	30: (* wait for com cycle *)
		IF NOT StartJob(TRUE) THEN // Not Busy, Execute set to True
			IF Error
			THEN
				ErrorText									:= CONCAT('Error at SlaveNo: ',	CONCAT(INT_TO_STRING(SlaveNo), CONCAT(', JobNo: ', INT_TO_STRING(JobNo))));
				SlaveCom[SlaveNo]^.countBad 				:= SlaveCom[SlaveNo]^.countBad +1;
				SlaveInErrorMask							:= CSETBIT32(SlaveInErrorMask,TO_SINT(SlaveNo),TRUE);
				IF Options.0
				THEN
					JobNo 									:= JobNo + 1;
					state 									:= 10;	(* next job *)				
				ELSE
					state 									:= 98; 					
				END_IF
			ELSE
				SlaveInErrorMask							:= CSETBIT32(SlaveInErrorMask,TO_SINT(SlaveNo),FALSE);
				SlaveCom[SlaveNo]^.countGood 				:= SlaveCom[SlaveNo]^.countGood +1;
				SlaveCom[SlaveNo]^.Jobs[JobNo].Valid 		:= TRUE;
				SlaveCom[SlaveNo]^.Jobs[JobNo].TimeStamp 	:= Timestamp;
				JobNo 										:= JobNo + 1;
				state 										:= 10;	(* next job *)
			END_IF
			StartJob(FALSE);
		END_IF

	98: (* wait for quit *)
		;


	END_CASE

METHOD PRIVATE getNextJob : Bool //Return value = TRUE if execution finished
VAR_INPUT
END_VAR
	
	WHILE SlaveCom[SlaveNo]^.Jobs[JobNo].FunctionCode = 0 DO
		JobNo 											:= JobNo + 1;
		IF JobNo > SlaveCom[SlaveNo]^.MAX_SLAVE_JOB THEN
			JobNo 										:= SlaveCom[SlaveNo]^.MIN_SLAVE_JOB;
			SlaveNo 									:= SlaveNo + 1;
			GetNextJob									:= FALSE;
			RETURN;
		END_IF
	END_WHILE
	GetNextJob											:= TRUE;
END_METHOD

METHOD PRIVATE getNextSlave : Bool //Return value = TRUE if execution finished
VAR_INPUT
END_VAR
	WHILE SlaveCom[SlaveNo] = 0 OR_ELSE NOT SlaveCom[SlaveNo]^.Enable DO
		SlaveNo 										:= SlaveNo + 1;
		IF SlaveNo > MAX_SLAVE 
		THEN
			k 											:= k + 1;
			SlaveNo 									:= MIN_SLAVE;
		ELSIF k = 2 
		THEN
			k 											:= 0;
			GetNextSlave								:= FALSE;
			RETURN;
		END_IF	
	END_WHILE
	GetNextSlave										:= TRUE;
END_METHOD

METHOD PUBLIC reset : BOOL //Return value = TRUE if execution finished
VAR_INPUT
END_VAR
IF State = 98 
THEN
	state													:= 0;
END_IF
Error														:= FALSE;
ErrorID														:= 0;
ErrorText													:= '';
reset														:= TRUE;
END_METHOD

METHOD PRIVATE startJob : BOOL //Return value = TRUE if busy - TRUE as long as the job is busy
VAR_INPUT
	Execute							: BOOL;
END_VAR
(* ModbusCOM Baustein mit parametern antriggern *)
	IF 	SlaveCom[SlaveNo]^.Jobs[JobNo].FunctionCode = 1 THEN
		com.ReadCoils(
			UnitID			:= SlaveCom[SlaveNo]^.Address,					(*UnitID: Modbus Stationsadresse (1..247). Der Modbus-Slave antwortet nur, wenn er Telegramme mit seiner eigenen Stationsadresse empfängt. optional können hier auch Sammeladressen eingestellt werden um auf beliebige Anfragen zu antworten. Die Adresse 0 ist für Broadcast-Telegramme reserviert und somit keine gültige Stationsadresse.*)
			Quantity		:= SlaveCom[SlaveNo]^.jobs[JobNo].Quantity,		(*Quantity: Anzahl der zu lesenden oder zu schreibenden Datenworte bei Wort-orientierten Modbus-Funktionen. Bei Bit-orientierten Modbus-Funktionen gibt Quantity die Anzahl der Bits (Inputs oder Coils) an.*)
			MBAddr			:= SlaveCom[SlaveNo]^.jobs[JobNo].startAddress,	(*MBAddr: Modbus-Datenadresse, von der die Daten aus dem Endgerät (Slave) gelesen werden. Diese Adresse wird unverändert zum Slave übertragen und wird dort als Datenadresse interpretiert.*)
			cbLength		:= SlaveCom[SlaveNo]^.jobs[JobNo].Quantity, 	(*cbLength : Größe der verwendeten Datenvariable für Sende- oder Lese-Aktionen in Bytes. cbLength muss größer oder gleich der durch Quantity bestimmten übertragenen Datenmenge sein. Bei Wortzugriffen gilt z. B.: [cbLength >= Quantity * 2]. cbLength kann mit SIZEOF(ModbusDaten) berechnet werden.*)
			pMemoryAddr		:= ADR(SlaveCom[SlaveNo]^.Data),				(*pMemoryAddr: Speicheradresse in der SPS, die mit ADR(ModbusDaten) berechnet wird. Bei Leseaktionen werden die gelesenen Daten in der adressierten Variablen abgelegt. Bei Sende-Aktionen werden die Daten aus der adressierten Variablen zum Endgerät übertragen.*)
			Execute			:= Execute,
			Timeout			:= ,
			BUSY			=> StartJob,									(*Busy: Zeigt an, dass der Funktionsbaustein aktiv ist. Busy wird mit steigender Flanke an Execute TRUE und wird wieder FALSE nachdem die gestartete Aktion beendet ist. Es kann immer nur eine Aktion gleichzeitig aktiv sein.*)
			Error			=> Error,										(*Error: Zeigt an, dass bei der Bearbeitung einer Aktion ein Fehler aufgetreten ist*)
			ErrorId			=> ErrorID);									(*ErrorId: Zeigt eine Fehlernummer im Falle einer gestörten oder fehlerhaften Kommunikation an.*)	

	ELSIF 	SlaveCom[SlaveNo]^.Jobs[JobNo].FunctionCode = 3 THEN
		com.ReadRegs(
			UnitID			:= SlaveCom[SlaveNo]^.Address,		
			Quantity		:= SlaveCom[SlaveNo]^.jobs[JobNo].Quantity,
			MBAddr			:= SlaveCom[SlaveNo]^.jobs[JobNo].startAddress,
			cbLength		:= SlaveCom[SlaveNo]^.jobs[JobNo].Quantity * 2,
			pMemoryAddr		:= ADR(SlaveCom[SlaveNo]^.data),
			Execute			:= Execute,
			Timeout			:= ,
			BUSY			=> StartJob,
			Error			=> Error,
			ErrorId			=> ErrorID);
	
	ELSIF 	SlaveCom[SlaveNo]^.Jobs[JobNo].FunctionCode = 4 THEN
		com.ReadInputRegs(
			UnitID			:= SlaveCom[SlaveNo]^.Address,		
			Quantity		:= SlaveCom[SlaveNo]^.jobs[JobNo].Quantity,
			MBAddr			:= SlaveCom[SlaveNo]^.jobs[JobNo].startAddress,
			cbLength		:= SlaveCom[SlaveNo]^.jobs[JobNo].Quantity * 2,
			pMemoryAddr		:= ADR(SlaveCom[SlaveNo]^.data),
			Execute			:= Execute,
			Timeout			:= ,
			BUSY			=> StartJob,
			Error			=> Error,
			ErrorId			=> ErrorID);
	
	ELSIF 	SlaveCom[SlaveNo]^.Jobs[JobNo].FunctionCode = 5 THEN
		com.WriteSingleCoil(
			UnitID			:= SlaveCom[SlaveNo]^.Address,		
			Quantity		:= SlaveCom[SlaveNo]^.jobs[JobNo].Quantity,
			MBAddr			:= SlaveCom[SlaveNo]^.jobs[JobNo].startAddress,
			cbLength		:= SlaveCom[SlaveNo]^.jobs[JobNo].Quantity,
			pMemoryAddr		:= ADR(SlaveCom[SlaveNo]^.data),
			Execute			:= Execute,
			Timeout			:= ,
			BUSY			=> StartJob,
			Error			=> Error,
			ErrorId			=> ErrorID);
			
	ELSIF 	SlaveCom[SlaveNo]^.Jobs[JobNo].FunctionCode = 6 THEN
		com.WriteSingleRegister(
			UnitID			:= SlaveCom[SlaveNo]^.Address,		
			Quantity		:= SlaveCom[SlaveNo]^.jobs[JobNo].Quantity,
			MBAddr			:= SlaveCom[SlaveNo]^.jobs[JobNo].startAddress,
			cbLength		:= SlaveCom[SlaveNo]^.jobs[JobNo].Quantity,
			pMemoryAddr		:= ADR(SlaveCom[SlaveNo]^.data),
			Execute			:= Execute,
			Timeout			:= ,
			BUSY			=> StartJob,
			Error			=> Error,
			ErrorId			=> ErrorID);
		
	ELSIF 	SlaveCom[SlaveNo]^.Jobs[JobNo].FunctionCode = 8 THEN
		com.Diagnostics(
			UnitID			:= SlaveCom[SlaveNo]^.Address,		
			Quantity		:= SlaveCom[SlaveNo]^.jobs[JobNo].Quantity,
			MBAddr			:= SlaveCom[SlaveNo]^.jobs[JobNo].startAddress,
			cbLength		:= SlaveCom[SlaveNo]^.jobs[JobNo].Quantity,
			pMemoryAddr		:= ADR(SlaveCom[SlaveNo]^.data),
			Execute			:= Execute,
			Timeout			:= ,
			BUSY			=> StartJob,
			Error			=> Error,
			ErrorId			=> ErrorID);
		
	ELSIF 	SlaveCom[SlaveNo]^.Jobs[JobNo].FunctionCode = 15 THEN
		com.WriteMultipleCoils(
			UnitID			:= SlaveCom[SlaveNo]^.Address,		
			Quantity		:= SlaveCom[SlaveNo]^.jobs[JobNo].Quantity,
			MBAddr			:= SlaveCom[SlaveNo]^.jobs[JobNo].startAddress,
			cbLength		:= SlaveCom[SlaveNo]^.jobs[JobNo].Quantity,
			pMemoryAddr		:= ADR(SlaveCom[SlaveNo]^.data),
			Execute			:= Execute,
			Timeout			:= ,
			BUSY			=> StartJob,
			Error			=> Error,
			ErrorId			=> ErrorID);
	
	ELSIF 	SlaveCom[SlaveNo]^.Jobs[JobNo].FunctionCode = 16 THEN
		com.WriteRegs(
			UnitID			:= SlaveCom[SlaveNo]^.Address,		
			Quantity		:= SlaveCom[SlaveNo]^.jobs[JobNo].Quantity,
			MBAddr			:= SlaveCom[SlaveNo]^.jobs[JobNo].startAddress,
			cbLength		:= SlaveCom[SlaveNo]^.jobs[JobNo].Quantity,
			pMemoryAddr		:= ADR(SlaveCom[SlaveNo]^.data),
			Execute			:= Execute,
			Timeout			:= ,
			BUSY			=> StartJob,
			Error			=> Error,
			ErrorId			=> ErrorID);
			
	END_IF
END_METHOD

END_FUNCTION_BLOCK

// ---- POUs/Connectivity/TF625x-Modbus/Master/TF6255-ModbusRtu/ModbusRtuMaster5B.TcPOU
{attribute 'no_check'}
// ModBus comunication master to multible slaves useing RTU protocol
// based on TF6255 - required lib: Tc2_ModbusRTU
FUNCTION_BLOCK ModbusRtuMaster5B
VAR_OUTPUT CONSTANT
	MIN_SLAVE												:	INT := 1;
	MAX_SLAVE												:	INT := PARAM.MODBUS_MAX_SLAVES_OF_MASTER;
{attribute 'displaymode':='binary'}
	OPTION_DISABLE_ERROR_STATE								:	BYTE := 2#0000_0001; //FB will not go into error state and keeps running, even all slaves are in error state
END_VAR
VAR_INPUT
	Enable													:	BOOL ; 		// FB will be processed as long as enable is TRUE 
	ResetTrig												:	BOOL ;		// The function block will be reset with a rising edge 
{attribute 'displaymode':='binary'}
	Options													:	BYTE := 0; //FB options, see VAR_OUTPUT CONSTANT
	SlaveCom												:	ARRAY[MIN_SLAVE..MAX_SLAVE] OF POINTER TO ModbusSlaveCom;
	Timestamp												:	DT;
END_VAR         	
VAR_OUTPUT     
	JobNo													:	INT := 0;
	SlaveNo													:	INT := 0;
{attribute 'displaymode':='binary'}
	SlaveInErrorMask										:	DWORD; //Bit.1 indicates slave 1 in error 	
	Error													:	BOOL;		// Rising edge of Error informs that an error occurred during the execution of the Function Block 
{attribute 'displaymode':='hex'}
	ErrorID													:	MODBUS_ERRORS;		// Error identification - see ADS return codes at Beckhoff infosys for further information 
	ErrorText												:	STRING;
END_VAR
VAR
(* memory **************************************************)
	State 													:	INT := 0;

(* trigger *************************************************)

(* timer ***************************************************)

(* blocks **************************************************)
//	com														:	ModbusRtuMaster_PcCOM := (Timeout := DEFAULT_ADS_TIMEOUT);
//	com														:	ModbusRtuMaster_KL6x22B := (Timeout := DEFAULT_ADS_TIMEOUT);
	com														:	ModbusRtuMaster_KL6x5B := (Timeout := DEFAULT_ADS_TIMEOUT);
(* internal used variables *********************************)
	i,j,k													:	INT :=0;
END_VAR

(* ModBus RTU comunication to multible slaves 	JHue V1.0			*)
(* uncomment necessary master funktion block 						*)
(* use TC2_ModBusRTU.lib											*)
(********************************************************************)
	IF ResetTrig THEN
		reset();
	END_IF
	
	CASE state OF
	0:	(* Idle *)
		IF Enable 
		THEN
			k 												:=	0;
			JobNo  :=  SlaveNo								:=	1;
			state 											:=	10;
		END_IF

	10: 
		IF GetNextSlave() 
		THEN (* find Slave *)
			k 												:= 0;
			IF GetNextJob() 
			THEN (* find JobNo *)
				SlaveCom[SlaveNo]^.currentJobIdx 			:= JobNo;
				SlaveCom[SlaveNo]^.writeJobRequested 		:= SlaveCom[SlaveNo]^.Jobs[JobNo].FunctionCode >= 5;
				State 										:= SEL(SlaveCom[SlaveNo]^.writeJobRequested, 20, 15);
			END_IF
		ELSE
			state 											:=	0;
		END_IF
	
	15: (* wait for valid write date *)
		IF NOT SlaveCom[SlaveNo]^.writeJobRequested
		THEN
			SlaveCom[SlaveNo]^.Jobs[JobNo].Valid 			:= FALSE;
			state 											:= 20;
		END_IF

	20: (* start job *)	
		IF NOT StartJob(FALSE) // Busy
		THEN						
			state 											:= 30;
		END_IF

	30: (* wait for com cycle *)
		IF NOT StartJob(TRUE) THEN // Not Busy, Execute set to True
			IF Error
			THEN
				ErrorText									:= CONCAT('Error at SlaveNo: ',	CONCAT(INT_TO_STRING(SlaveNo), CONCAT(', JobNo: ', INT_TO_STRING(JobNo))));
				SlaveCom[SlaveNo]^.countBad 				:= SlaveCom[SlaveNo]^.countBad +1;
				SlaveInErrorMask							:= CSETBIT32(SlaveInErrorMask,TO_SINT(SlaveNo),TRUE);
				IF Options.0
				THEN
					JobNo 									:= JobNo + 1;
					state 									:= 10;	(* next job *)				
				ELSE
					state 									:= 98; 					
				END_IF
			ELSE
				SlaveInErrorMask							:= CSETBIT32(SlaveInErrorMask,TO_SINT(SlaveNo),FALSE);
				SlaveCom[SlaveNo]^.countGood 				:= SlaveCom[SlaveNo]^.countGood +1;
				SlaveCom[SlaveNo]^.Jobs[JobNo].Valid 		:= TRUE;
				SlaveCom[SlaveNo]^.Jobs[JobNo].TimeStamp 	:= Timestamp;
				JobNo 										:= JobNo + 1;
				state 										:= 10;	(* next job *)
			END_IF
			StartJob(FALSE);
		END_IF

	98: (* wait for quit *)
		;


	END_CASE

METHOD PRIVATE getNextJob : Bool
VAR_INPUT
END_VAR
	
	WHILE SlaveCom[SlaveNo]^.Jobs[JobNo].FunctionCode = 0 DO
		JobNo 											:= JobNo + 1;
		IF JobNo > SlaveCom[SlaveNo]^.MAX_SLAVE_JOB THEN
			JobNo 										:= SlaveCom[SlaveNo]^.MIN_SLAVE_JOB;
			SlaveNo 									:= SlaveNo + 1;
			GetNextJob									:= FALSE;
			RETURN;
		END_IF
	END_WHILE
	GetNextJob											:= TRUE;
END_METHOD

METHOD PRIVATE getNextSlave : Bool
VAR_INPUT
END_VAR
	WHILE SlaveCom[SlaveNo] = 0 OR_ELSE NOT SlaveCom[SlaveNo]^.Enable DO
		SlaveNo 										:= SlaveNo + 1;
		IF SlaveNo > MAX_SLAVE 
		THEN
			k 											:= k + 1;
			SlaveNo 									:= MIN_SLAVE;
		ELSIF k = 2 
		THEN
			k 											:= 0;
			GetNextSlave								:= FALSE;
			RETURN;
		END_IF	
	END_WHILE
	GetNextSlave										:= TRUE;
END_METHOD

METHOD PUBLIC reset : booL //Return value = TRUE if execution finished
VAR_INPUT
END_VAR
IF State = 98 
THEN
	state													:= 0;
END_IF
Error														:= FALSE;
ErrorID														:= 0;
ErrorText													:= '';
reset														:= TRUE;
END_METHOD

METHOD PRIVATE startJob : BOOL //Return value = TRUE if busy - TRUE as long as the job is busy
VAR_INPUT
	Execute							: BOOL;
END_VAR
(* ModbusCOM Baustein mit parametern antriggern *)
	IF 		SlaveCom[SlaveNo]^.Jobs[JobNo].FunctionCode = 1 THEN
		com.ReadCoils(
			UnitID			:= SlaveCom[SlaveNo]^.Address,				(*UnitID: Modbus Stationsadresse (1..247). Der Modbus-Slave antwortet nur, wenn er Telegramme mit seiner eigenen Stationsadresse empfängt. optional können hier auch Sammeladressen eingestellt werden um auf beliebige Anfragen zu antworten. Die Adresse 0 ist für Broadcast-Telegramme reserviert und somit keine gültige Stationsadresse.*)
			Quantity		:= SlaveCom[SlaveNo]^.jobs[JobNo].Quantity,		(*Quantity: Anzahl der zu lesenden oder zu schreibenden Datenworte bei Wort-orientierten Modbus-Funktionen. Bei Bit-orientierten Modbus-Funktionen gibt Quantity die Anzahl der Bits (Inputs oder Coils) an.*)
			MBAddr			:= SlaveCom[SlaveNo]^.jobs[JobNo].startAddress,	(*MBAddr: Modbus-Datenadresse, von der die Daten aus dem Endgerät (Slave) gelesen werden. Diese Adresse wird unverändert zum Slave übertragen und wird dort als Datenadresse interpretiert.*)
			cbLength		:= SlaveCom[SlaveNo]^.jobs[JobNo].Quantity, 	(*cbLength : Größe der verwendeten Datenvariable für Sende- oder Lese-Aktionen in Bytes. cbLength muss größer oder gleich der durch Quantity bestimmten übertragenen Datenmenge sein. Bei Wortzugriffen gilt z. B.: [cbLength >= Quantity * 2]. cbLength kann mit SIZEOF(ModbusDaten) berechnet werden.*)
			pMemoryAddr		:= ADR(SlaveCom[SlaveNo]^.Data),				(*pMemoryAddr: Speicheradresse in der SPS, die mit ADR(ModbusDaten) berechnet wird. Bei Leseaktionen werden die gelesenen Daten in der adressierten Variablen abgelegt. Bei Sende-Aktionen werden die Daten aus der adressierten Variablen zum Endgerät übertragen.*)
			Execute			:= Execute,
			Timeout			:= ,
			BUSY			=> StartJob,									(*Busy: Zeigt an, dass der Funktionsbaustein aktiv ist. Busy wird mit steigender Flanke an Execute TRUE und wird wieder FALSE nachdem die gestartete Aktion beendet ist. Es kann immer nur eine Aktion gleichzeitig aktiv sein.*)
			Error			=> Error,										(*Error: Zeigt an, dass bei der Bearbeitung einer Aktion ein Fehler aufgetreten ist*)
			ErrorId			=> ErrorID);									(*ErrorId: Zeigt eine Fehlernummer im Falle einer gestörten oder fehlerhaften Kommunikation an.*)	
	
	ELSIF 	SlaveCom[SlaveNo]^.Jobs[JobNo].FunctionCode = 3 THEN
		com.ReadRegs(
			UnitID			:= SlaveCom[SlaveNo]^.Address,		
			Quantity		:= SlaveCom[SlaveNo]^.jobs[JobNo].Quantity,
			MBAddr			:= SlaveCom[SlaveNo]^.jobs[JobNo].startAddress,
			cbLength		:= SlaveCom[SlaveNo]^.jobs[JobNo].Quantity * 2,
			pMemoryAddr		:= ADR(SlaveCom[SlaveNo]^.data),
			Execute			:= Execute,
			Timeout			:= ,
			BUSY			=> StartJob,
			Error			=> Error,
			ErrorId			=> ErrorID);
	
	ELSIF 	SlaveCom[SlaveNo]^.Jobs[JobNo].FunctionCode = 4 THEN
		com.ReadInputRegs(
			UnitID			:= SlaveCom[SlaveNo]^.Address,		
			Quantity		:= SlaveCom[SlaveNo]^.jobs[JobNo].Quantity,
			MBAddr			:= SlaveCom[SlaveNo]^.jobs[JobNo].startAddress,
			cbLength		:= SlaveCom[SlaveNo]^.jobs[JobNo].Quantity * 2,
			pMemoryAddr		:= ADR(SlaveCom[SlaveNo]^.data),
			Execute			:= Execute,
			Timeout			:= ,
			BUSY			=> StartJob,
			Error			=> Error,
			ErrorId			=> ErrorID);
	
	ELSIF 	SlaveCom[SlaveNo]^.Jobs[JobNo].FunctionCode = 5 THEN
		com.WriteSingleCoil(
			UnitID			:= SlaveCom[SlaveNo]^.Address,		
			Quantity		:= SlaveCom[SlaveNo]^.jobs[JobNo].Quantity,
			MBAddr			:= SlaveCom[SlaveNo]^.jobs[JobNo].startAddress,
			cbLength		:= SlaveCom[SlaveNo]^.jobs[JobNo].Quantity,
			pMemoryAddr		:= ADR(SlaveCom[SlaveNo]^.data),
			Execute			:= Execute,
			Timeout			:= ,
			BUSY			=> StartJob,
			Error			=> Error,
			ErrorId			=> ErrorID);
		
	ELSIF 	SlaveCom[SlaveNo]^.Jobs[JobNo].FunctionCode = 6 THEN
		com.WriteSingleRegister(
			UnitID			:= SlaveCom[SlaveNo]^.Address,		
			Quantity		:= SlaveCom[SlaveNo]^.jobs[JobNo].Quantity,
			MBAddr			:= SlaveCom[SlaveNo]^.jobs[JobNo].startAddress,
			cbLength		:= SlaveCom[SlaveNo]^.jobs[JobNo].Quantity,
			pMemoryAddr		:= ADR(SlaveCom[SlaveNo]^.data),
			Execute			:= Execute,
			Timeout			:= ,
			BUSY			=> StartJob,
			Error			=> Error,
			ErrorId			=> ErrorID);
			
	ELSIF 	SlaveCom[SlaveNo]^.Jobs[JobNo].FunctionCode = 8 THEN
		com.Diagnostics(
			UnitID			:= SlaveCom[SlaveNo]^.Address,		
			Quantity		:= SlaveCom[SlaveNo]^.jobs[JobNo].Quantity,
			MBAddr			:= SlaveCom[SlaveNo]^.jobs[JobNo].startAddress,
			cbLength		:= SlaveCom[SlaveNo]^.jobs[JobNo].Quantity,
			pMemoryAddr		:= ADR(SlaveCom[SlaveNo]^.data),
			Execute			:= Execute,
			Timeout			:= ,
			BUSY			=> StartJob,
			Error			=> Error,
			ErrorId			=> ErrorID);
	
	ELSIF 	SlaveCom[SlaveNo]^.Jobs[JobNo].FunctionCode = 15 THEN
		com.WriteMultipleCoils(
			UnitID			:= SlaveCom[SlaveNo]^.Address,		
			Quantity		:= SlaveCom[SlaveNo]^.jobs[JobNo].Quantity,
			MBAddr			:= SlaveCom[SlaveNo]^.jobs[JobNo].startAddress,
			cbLength		:= SlaveCom[SlaveNo]^.jobs[JobNo].Quantity,
			pMemoryAddr		:= ADR(SlaveCom[SlaveNo]^.data),
			Execute			:= Execute,
			Timeout			:= ,
			BUSY			=> StartJob,
			Error			=> Error,
			ErrorId			=> ErrorID);
	
	ELSIF 	SlaveCom[SlaveNo]^.Jobs[JobNo].FunctionCode = 16 THEN
		com.WriteRegs(
			UnitID			:= SlaveCom[SlaveNo]^.Address,		
			Quantity		:= SlaveCom[SlaveNo]^.jobs[JobNo].Quantity,
			MBAddr			:= SlaveCom[SlaveNo]^.jobs[JobNo].startAddress,
			cbLength		:= SlaveCom[SlaveNo]^.jobs[JobNo].Quantity,
			pMemoryAddr		:= ADR(SlaveCom[SlaveNo]^.data),
			Execute			:= Execute,
			Timeout			:= ,
			BUSY			=> StartJob,
			Error			=> Error,
			ErrorId			=> ErrorID);	
	END_IF
END_METHOD

END_FUNCTION_BLOCK

// ---- POUs/Connectivity/TF6310-TcpServer/TcpBasic/TCPSendRecCtrl.TcPOU
{attribute 'no_check'}
//Send or receive data via TCP connection 
//based on TF6310, required lib: Tc2_TcpIp - see Beckhoff Infosys for more information
FUNCTION_BLOCK TCPSendRecCtrl EXTENDS FbBase
VAR_OUTPUT CONSTANT
	FNC_RECEIVE												:	INT := 0;
	FNC_SEND												:	INT := 1;
END_VAR                 									
VAR_INPUT               									
	Fnc														:	INT (FNC_RECEIVE..FNC_SEND) := FNC_RECEIVE;
	SrvNetId												: 	T_AmsNetId := ''; (* server ams net id *)
	Timeout													: 	TIME := DEFAULT_ADS_TIMEOUT; //ADS timeout
{attribute 'displaymode':='binary'}
	Options													:	BYTE := 2#0000_0000; //Options Bit .0 = Do NOT restart receive internally
	hSocket													:	T_HSOCKET; //Server handle
	pData													:	POINTER TO BYTE; //Pointer do send/res data field 
	cbData													:	UDINT; //Size of send/rec data field 
	EnableDebugMode											:	BOOL; //Write debug information into twincat logger
END_VAR
VAR_OUTPUT
	RecBytes 												:  UDINT;  	// Count of received bytes
	WinsockErrorId											:	E_WinsockError;  //Winsocket error enum - see TF6310 documentation for further information
END_VAR
VAR
(* cache ************************************************************)
	MemFnc													:	INT := -1;

(* function-block instances ***************************************************************)
	SocketSend												:	FB_SocketSend;
	SocketReceive											:	FB_SocketReceive;

END_VAR


(* Execute ***************************************************************************************)
	rtExecute(CLK := Execute);
	IF rtExecute.Q
		AND MemFnc < 0
	THEN
		MemFnc 												:= SEL(Fnc = FNC_SEND, FNC_RECEIVE , FNC_SEND) ;
		Busy												:= TRUE;
		Done												:= FALSE;
		Error												:= FALSE;
		ErrorID												:= 0;
	END_IF

(* Call Method ***********************************************************************************)
	CASE MemFnc OF
	FNC_SEND:
		SEND(Execute:= Execute);

	FNC_RECEIVE:
		Receive(Execute	:= Execute);

	-1:
		IF NOT Execute
		THEN
			Busy											:= FALSE;
			Done											:= FALSE;
			Error											:= FALSE;
			ErrorID											:= 0;
		END_IF                              				
	ELSE                                    				
		Busy												:= FALSE;
		Done												:= FALSE;
		Error												:= Execute;
		ErrorID												:= E_AdsErr.DEVICE_INVALIDPARM;
	END_CASE

(*************************************************************************************************)

PROPERTY PUBLIC optDoNotRestartReceiveCyclic : BOOL
GET
optDoNotRestartReceiveCyclic := Options.0;
END_GET
SET
Options.0 := optDoNotRestartReceiveCyclic;
END_SET
END_PROPERTY

METHOD PUBLIC receive : BOOL //Return value = TRUE if busy
//required parameter
//hSocket
//pData
//cbData
VAR_INPUT
	Execute													:	BOOL;
END_VAR
	MemFnc													:= FNC_RECEIVE;
	THIS^.Execute											:= Execute;
	                                						
IF pData = 0                        						
THEN                                						
	Busy													:= NOT Error;
	Error													:= TRUE;
	ErrorId													:= E_AdsErr.DEVICE_INVALIDPARM;
	Done													:= FALSE;
	MemFnc													:= SEL(Execute , -1 ,MemFnc); 
	RETURN;                         	
END_IF

	IF Execute
	THEN
		Error												:=	FALSE;
		ErrorId												:= 0;
		SocketReceive.bExecute 								:= TRUE;
	ELSIF NOT SocketReceive.bBusy   						
	THEN                            						
		Error												:=	FALSE;
		ErrorId												:= 0;
		SocketReceive.bExecute 								:= FALSE;
	END_IF                          	
                                    	
	SocketReceive(
			sSrvNetId	:= SrvNetId,
			hSocket		:= hSocket,
			cbLen		:= cbData,
			pDest		:= pData,
			bExecute	:= ,
			tTimeout	:= Timeout,
			bBusy		=> Busy,
			bError		=> ,
			nErrId		=> ,
			nRecBytes	=> );

	IF NOT SocketReceive.bBusy
		AND NOT SocketReceive.bError
		AND SocketReceive.bExecute
	THEN
		IF EnableDebugMode
			AND SocketReceive.nRecBytes > 0
			AND NOT Done
		THEN
			ADSLOGDINT(	ADSLOG_MSGTYPE_ERROR OR ADSLOG_MSGTYPE_LOG, CONCAT('%d Bytes received / ', HSOCKET_TO_STRING(hSocket)) , UDINT_TO_DINT(SocketReceive.nRecBytes));
		END_IF
		Done												:= SocketReceive.nRecBytes > 0 OR Options.0; (* Done melden nach jedenm Lesezyklus, egal ob Daten empfangen wurden *)
		IF NOT Done
		THEN (* only set Done if something is safely received *)
			SocketReceive(bExecute := FALSE);
			SocketReceive(bExecute := TRUE, bBusy => Busy);
		END_IF
		RecBytes											:= SEL(Done , 0 ,SocketReceive.nRecBytes);
	ELSE                                					
		Done												:= FALSE;
	END_IF                              	
                                        	
	IF NOT Busy
	THEN
		IF SocketReceive.bExecute
		THEN
			Error											:=	SocketReceive.bError;
			IF SocketReceive.nErrId >= 16#80070000
			THEN
				ErrorId										:= E_ADSERR.CLIENT_W32ERROR;
				WinsockErrorId								:= ADSERROR_TO_WSERROR(SocketReceive.nErrId);
			ELSE                    						
				ErrorId										:= SocketReceive.nErrId;
				WinsockErrorId								:= WSOK;
			END_IF
		END_IF
		IF NOT Execute
		THEN
			MemFnc											:= -1;
			SocketReceive(bExecute := FALSE);
		END_IF
	END_IF
	
	//Method return
	Receive													:= Busy;
END_METHOD

METHOD PUBLIC send : BOOL //Return value = TRUE if busy
//required parameter
//hSocket
//pData
//cbData
VAR_INPUT
	Execute													:	BOOL;
END_VAR
	MemFnc													:= FNC_SEND;
	THIS^.Execute											:= Execute;
	
IF pData = 0 THEN
	Busy													:= NOT Error;
	Error													:= TRUE;
	ErrorId													:= E_ADSErr.DEVICE_INVALIDPARM;
	Done													:= FALSE;
	MemFnc													:= SEL(Execute , -1 ,MemFnc); 
	RETURN;
END_IF

	IF Execute
	THEN
		Error												:=	FALSE;
		ErrorId												:= 0;
		SocketSend.bExecute 								:= TRUE;
	ELSIF NOT SocketSend.bBusy          					
	THEN                                					
		Error												:=	FALSE;
		ErrorId												:= 0;
		SocketSend.bExecute 								:= FALSE;
	END_IF                              	
	                                    	
	SocketSend(
		sSrvNetId	:= SrvNetId,
		hSocket		:= hSocket,
		cbLen		:= cbData,
		pSrc		:= pData,
		bExecute	:= ,
		tTimeout	:= Timeout,
		bBusy		=> Busy,
		bError		=> ,
		nErrId		=> );

	IF NOT SocketSend.bBusy
		AND NOT SocketSend.bError
		AND SocketSend.bExecute
	THEN
		IF NOT Done
			AND EnableDebugMode
		THEN
			ADSLOGDINT(	ADSLOG_MSGTYPE_ERROR OR ADSLOG_MSGTYPE_LOG, CONCAT('%d Bytes sended / ', HSOCKET_TO_STRING(hSocket)) , UDINT_TO_DINT(cbData));
		END_IF
		Done												:= TRUE;
	ELSE                                					
		Done												:= FALSE;
	END_IF

	IF NOT Busy
	THEN
		IF SocketSend.bExecute
		THEN
			Error											:=	SocketSend.bError;
			IF SocketSend.nErrId >= 16#80070000
			THEN
				ErrorId										:= E_AdsErr.CLIENT_W32ERROR;
				WinsockErrorId								:= ADSERROR_TO_WSERROR(SocketSend.nErrId);
			ELSE
				ErrorId										:= SocketSend.nErrId;
				WinsockErrorId								:= WSOK;
			END_IF
		END_IF
		IF NOT Execute
		THEN
			MemFnc											:= -1;
			SocketSend(bExecute := FALSE);
		END_IF
	END_IF
	
	//Method return
	Send													:= Busy;
END_METHOD

END_FUNCTION_BLOCK

// ---- POUs/Connectivity/TF6310-TcpServer/UdpBasic/UDPServerCtrl.TcPOU
{attribute 'no_check'}
//Helper for UDP Client or Server for socket communications. (Wrapper for Fbs like SocketAccpet,SocketClose,SocketConnect....)
//based on TF6310, required lib: Tc2_TcpIp - see Beckhoff Infosys for more information
FUNCTION_BLOCK UDPServerCtrl 
VAR_INPUT
	Enable													:	BOOL := FALSE;	// FB will be processed as long as enable is TRUE 
	SrvNetId												: 	T_AmsNetId := ''; 	// AmsNet id for TcpIp Server instance - '' for local 
	SrvLocalHost											:	T_IPv4Addr := ''; 	// IP-Adress of local ip-adapter used for server communication
	SrvLocalPort											:	UDINT;			//	IP-Port of local ip-adapter used for server communication

	EnableDebugMode											:	BOOL := FALSE; 	// Write debug information into twincat logger
	CloseAllSocket											:	BOOL := TRUE; 	// Close all socket if server will be diabled - FALSE = close only connected port
END_VAR
VAR_OUTPUT
	hSocket													: 	T_HSOCKET ;	// UDP socket handle
	Online													:	BOOL; 	// Connection is current running 
	State													:	E_SocketConnectionState; //Socket connection state enum
	Busy													:	BOOL;	// Busy is TRUE at the rising edge of Enable and stays TRUE as long as the FB is performing any action. 
	Error													:	BOOL;	// Rising edge of Error informs that an error occurred during the execution of the Function Block #
{attribute 'displaymode':='hex'}
	ErrorId													:	UDINT; 	// Error identification - see ADS return codes and TF6310 documentation at Beckhoff infosys for further information
	WinsockErrorId											:	E_WinsockError; // Winsocket error enum - see TF6310 documentation for further information
END_VAR
VAR
(* function-block instances ***************************************************************)
	SocketCtrl												:	UDPSocketCtrl;

END_VAR


(* Execute ****************************************************)
	SocketCtrl(
		Execute			:= ,
		Fnc				:= ,
		SrvNetId		:= '', (* Server IP *)
		LocalHost		:= SrvLocalHost, (* Own IP *)
		LocalPort		:= SrvLocalPort,
		Timeout			:= t#30s,
		Online			=> Online,
		hSocket			=> hSocket,
		Done			=> ,
		Busy			=> Busy,
		Error			=> Error,
		ErrorId			=> ErrorId,
		WinsockErrorId 	=> WinsockErrorId);

	IF Busy
	THEN
		SocketCtrl.Execute 									:= Enable;
	ELSIF SocketCtrl.Done
	THEN
		IF EnableDebugMode
		THEN
			ADSLOGDINT(	ADSLOG_MSGTYPE_ERROR OR ADSLOG_MSGTYPE_LOG, SocketCtrl.hSocketText, 0);
		END_IF
		SocketCtrl(Execute := FALSE);
		Busy												:= FALSE;
		Error												:= FALSE;
		ErrorId												:= 0;
		WinsockErrorId										:= WSOK;
	ELSIF SocketCtrl.Error
	THEN
		IF NOT Enable
		THEN
			SocketCtrl(Execute := FALSE);
			Busy											:= FALSE;
			Error											:= FALSE;
			ErrorId											:= 0;
			WinsockErrorId									:= WSOK;
		END_IF
	ELSE
		IF Enable
			AND NOT Online
		THEN
			SocketCtrl(Execute := FALSE);
			SocketCtrl.Execute 								:= TRUE;
			SocketCtrl.Fnc 									:= SocketCtrl.FNC_CREATE;
			Busy											:= TRUE;
			Error											:= FALSE;
			ErrorId											:= 0;
			WinsockErrorId									:= WSOK;

		ELSIF Online
			AND NOT Enable
		THEN
			SocketCtrl(Execute := FALSE);
			SocketCtrl.Execute 								:= TRUE;
			SocketCtrl.Fnc 									:= SEL(CloseAllSocket, SocketCtrl.FNC_CLOSE,  SocketCtrl.FNC_CLOSE_ALL);
			Busy											:= TRUE;
			Error											:= FALSE;
			ErrorId											:= 0;
			WinsockErrorId									:= WSOK;
		ELSE
			;
		END_IF
	END_IF

(******************************************************************************)

END_FUNCTION_BLOCK

// ---- POUs/ControllerTools/PIDController.TcPOU
//Base PID controller with manual 
FUNCTION_BLOCK PIDController 
VAR_INPUT
	Enable													: BOOL := FALSE;	// FB will be processed as long as enable is TRUE 
	ResetTrig												: BOOL := FALSE;	// The function block will get reseted with a rising edge 
	ManualOn												: BOOL := FALSE;	// set Q to ManualValue 
	Sync													: BOOL := FALSE;	// synchronization flag for bumpless initialisation
	// controller input (deviation)   					
	SetValue												: LREAL := 0.0;		// Setpoint value										
	ActValue												: LREAL := 0.0;		// Actual value											
	
	MinOutput												: LREAL := 0.0;		// controller minimum output (min. limit)				
	MaxOutput												: LREAL := 0.0;		// controller maximum output (max. limit)				
	SyncValue												: LREAL := 0.0;		// syncronization value for bumpless init.				
	ManualValue												: LREAL := 0.0;		// manual value *)
	// controller values             					
	CycleTime												: LREAL := 0.0;		// controller cycle time in seconds [s]					
	Kp														: LREAL := 0.0;		// proportional gain Kp	(P)								
	Tn														: LREAL := 0.0;		// integral gain Tn (I) [s]								
	Tv														: LREAL := 0.0;		// derivative gain Tv (D-T1) [s]						
	Td														: LREAL := 0.0;		// derivative damping time Td (D-T1) [s]				
	InnerWindow												: LREAL := 0.0;		// inner window for reduced I-part (dE-window)			
	OuterWindow												: LREAL := 0.0;		// outer window for disabling I-part (dE-window)		
END_VAR
VAR_OUTPUT
	Q														: LREAL := 0;		// controller output command							
	Deviation												: LREAL := 0.0;		// Setpoint deviation									
	MinLimit												: BOOL := FALSE;	// minimum limiting active ? [TRUE/FALSE] -> ARW		
	MaxLimit												: BOOL := FALSE;	// maximum limiting active ? [TRUE/FALSE] -> ARW		
	ARWActive												: BOOL := FALSE;	// ARW actice ? [TRUE/FALSE] -> freeze I-part			
	Error													: BOOL := FALSE;	// Rising edge of Error informs that an error occurred during the execution of the Function Block 							
	ErrorId													: UDINT := 0;		// Error identification 		
END_VAR                         							
VAR_OUTPUT CONSTANT                   							
	ERR_NOERROR												: UDINT := 0;		// no error												
	ERR_NOINIT												: UDINT := 1;		// no initialization done								
	ERR_INVALIDPARAM										: UDINT := 2;		// invalid parameter								
	ERR_INVALIDCYCLETIME									: UDINT := 3;		// invalid cycle time									
END_VAR
VAR
	// STATIC VARIABLE
	// Internal Variable
	fE														: LREAL := 0.0;		// error input											
	fE_1													: LREAL := 0.0;		// error input z^(-1)									
	fY														: LREAL := 0.0;		// control output										
	fY_1													: LREAL := 0.0;		// control output  z^(-1)								
	fYP														: LREAL := 0.0;		// P-part												
	fYI														: LREAL := 0.0;		// I-part												
	fYI_1													: LREAL := 0.0;		// I-part  z^(-1)										
	fYD														: LREAL := 0.0;		// D-T1-part										
	fYD_1													: LREAL := 0.0;		// D-T1-part  z^(-1)									
	// Internal Parameter
	bIsInitDone												: BOOL	:= FALSE;	// is controller init done ?							
	bInitMem												: BOOL	:= FALSE;	// reset flag											
	bIsIPart												: BOOL	:= FALSE;	// I-part active ?										
	bIsDPart												: BOOL	:= FALSE;	// D-part active ?										
	bIsDAutoScaling											: BOOL	:= FALSE;	// autoscaling for D-part done ?						
	bIsOuterWnd												: BOOL	:= FALSE;	// I-part active and outer window unequal zero ?		
                                							
	fDi														: LREAL	:= 0.0;		// internal I param										
	fDd														: LREAL	:= 0.0;		// internal D param										
	fCd														: LREAL	:= 0.0;		// internal D param										
	fCycleTime												: LREAL	:= 0.0;		// controller cycle time [s]
	MemSyncValue											: LREAL	:= 0.0;
	rtSync													: r_trig;
	rtReset													: r_trig;
END_VAR

(* controller init *)
rtReset(CLK := ResetTrig);
IF rtReset.Q OR NOT bIsInitDone OR NOT Enable 
THEN
	reset();
	RETURN;
END_IF

(* 1. check for initialisation flag *)
IF bIsInitDone 
THEN
	ErrorID 												:= ERR_NOERROR;
ELSE                                    					
	Error 													:= TRUE;
	ErrorID 												:= ERR_NOINIT;
END_IF

(* 2. controller synchronization flag => look at the end of FB *)
(* I-part *)
IF( Tn > 0.0 ) 
THEN
	fDi 												:= (Kp * fCycleTime) / (2.0 * Tn);
	bIsIPart											:= TRUE;
ELSE                                    				
	fDi 												:= 0.0;
	bIsIPart 											:= FALSE;
END_IF

(* D-part *)
IF	( Tv > 0.0 ) AND (Td > 0.0) 
THEN
	(* autoscaling necessary if (Td < CycleTime) or (Tv < Td)	*)
	(* if (Td < CycleTime) => (Td = CycleTime)					*)
	IF	( Td < fCycleTime ) 
	THEN(* autoscaling for D-part *)
		bIsDAutoScaling									:= TRUE;
		fDd 											:= (Kp * Tv) / (fCycleTime + fCycleTime / 2.0);
		fCd 											:= (fCycleTime / 2.0) / (fCycleTime + fCycleTime / 2.0);
	ELSE(* normal calculation, no autoscaling for D-part *)
		bIsDAutoScaling									:= FALSE;
		fDd 											:= (Kp * Tv) / (Td + fCycleTime / 2.0);
		fCd 											:= (Td - fCycleTime / 2.0) / (Td + fCycleTime / 2.0);
	END_IF;                             				
	bIsDPart 											:= TRUE;                   				
ELSE                                    				
	fDd													:= 0.0;
	fCd 												:= 0.0;
	bIsDPart 											:= FALSE;
END_IF;                                 				
                                        				
                                        				
(* 3. save old variable *)              				
fE_1													:= fE;
fY_1													:= fY;
fYI_1													:= fYI;
fYD_1													:= fYD;
                                        				
(* 4. set error/deviation input *)      				
Deviation												:= SetValue - ActValue;
fE														:= Deviation;  
                                     				
(* 5. YP-part *)                        	
fYp														:= Kp * fE;
                                        				
(* 6. YI-part *)                        				
IF bIsIPart                             				
THEN                                    				
	IF	( MinLimit                      				
		AND (fE < 0.0) )                				
	THEN                                				
		ARWActive										:= TRUE;
		fYI												:= fYI_1;						(* freeze I-part *)
	ELSIF	( MaxLimit                  				
			AND (fE > 0.0) )            				
	THEN                                				
		ARWActive										:= TRUE;
		fYI												:= fYI_1;						(* freeze I-part *)
	ELSE
		ARWActive										:= FALSE;
		(* fYI		:= fYI_1 + fDi * (fE + fE_1); *)					(* normal I-part calculation *)

		(* reduce I-part in the inner window *)
		IF ( ABS( fE ) < InnerWindow ) 
		THEN
			fYI 						:= fYI_1 + fDi * (fE + fE_1) * (ABS( fE ) / InnerWindow);(* reduced I-part *)
		ELSIF ( bIsOuterWnd AND ( ABS( fE ) > OuterWindow ) ) 
		THEN
			fYI											:= fYI_1;						(* freeze I-part in outer window *)
		ELSE                            				
			fYI 										:= fYI_1 + fDi * (fE + fE_1);	(* normal I-part calculation *)
		END_IF                          				
                                        				
	END_IF                              				
ELSE                                    				
	ARWActive											:= FALSE;
	fYI													:= 0.0;
END_IF                                  				
                                        	
(* 7. YD-part *)                        	
IF bIsDPart THEN                        	
	fYD													:=  fCd * fYD_1 + fDd * (fE - fE_1);
ELSE                                    				
	fYD													:= 0.0;
END_IF                                  				
                                        				
(* 8. Ysum = YP + YI + YD *)            				
fY														:= fYP + fYI + fYD;

(* 2. synchronization: Bumpless Init Without Abrupt Change Of Y(t) *)
rtSync(CLK := Sync);
IF 	ManualOn 
	OR rtSync.Q 
THEN
	Synchronize(SEL(ManualOn,SyncValue,ManualValue));
END_IF                                  				
                                        				
(* 9. check for output limiting *)      				
IF ( fY >= MaxOutput )                  				
THEN                                    				
	fY													:= MaxOutput;
	MinLimit											:= FALSE;
	MaxLimit											:= TRUE;
ELSIF ( fY <= MinOutput )               				
THEN                                    	
	fY													:= MinOutput;
	MinLimit											:= TRUE;
	MaxLimit											:= FALSE;
ELSE                                    				
	MinLimit											:= FALSE;
	MaxLimit											:= FALSE;
END_IF

(* 10. set controller output *)
Q 														:= fY;

(**********************************************************************************)

METHOD PUBLIC reset : BOOL; //Return value = TRUE if execution finished
VAR_INPUT
END_VAR
(* reset internal and external variables *)

fE															:= fE_1		:= 0.0;
fY															:= fY_1		:= 0.0;
fYP															:= 0.0;
fYI															:= fYI_1	:= 0.0;
fYD															:= fYD_1	:= 0.0;
bIsInitDone													:= FALSE;
bIsIPart													:= FALSE;
bIsDPart													:= FALSE;
ARWActive													:= FALSE;
bIsDAutoScaling												:= FALSE;
bIsOuterWnd													:= FALSE;
Q															:= 0.0;
MinLimit													:= FALSE;
MaxLimit													:= FALSE;
Error 														:= FALSE;
                            								
(* ??? set fE=fCtrlInput und fE_1=fCtrlInput ??? *)
(*	fE	:=  fCtrlInput; *)

(* read PLC cycle time for discreete calculation *)
(*	fCycleTime	:=	DINT_TO_REAL( GetScanTime( dummyInVar:= TRUE ) ) * 0.000001; *)
fCycleTime													:= CycleTime;

(* check cycle time parameter: (CycleTime > 0 AND CycleTme <= 60) *)
IF (fCycleTime <= 0) OR (fCycleTime > 60.0) 
THEN
	ErrorID 												:= ERR_INVALIDCYCLETIME;
	Error													:= TRUE;
	RETURN;
END_IF;

(* check controller parameters: (Tn, Tv, Td >= 0) *)
IF 	( (Tn < 0) 
	OR (Tv < 0) OR (Td < 0) ) 
THEN
	ErrorID 												:= ERR_INVALIDPARAM;
	Error													:= TRUE;
	RETURN;
END_IF;

(* check controller parameters: (MinOutput > MaxOutput) *)
IF ( MinOutput > MaxOutput ) 
THEN
	ErrorID 												:= ERR_INVALIDPARAM;
	Error													:= TRUE;
	RETURN;
END_IF;

(* check inner and outer window parameters: outer window must be greater than the inner window *)
IF((bIsIPart) AND ( OuterWindow > 0.0 )) 
THEN
	IF (InnerWindow > OuterWindow) 
	THEN
		ErrorId 											:= ERR_INVALIDPARAM;
		Error												:= TRUE;
		RETURN;
	END_IF;
	bIsOuterWnd 											:= TRUE;
END_IF;

(* set internal init flag *)
bIsInitDone													:= TRUE;
Q		 													:= MinOutput;
reset													:= TRUE;
END_METHOD

METHOD PUBLIC synchronize : BOOL  //Return value = TRUE if execution finished
VAR_INPUT 
	IN											:	LREAL;
END_VAR
	MemSyncValue										:= IN;
	
	(* Demand:  SyncValue != Ysum  with  SyncValue = Ysum = YP + YI + YD  =>  YI = SyncValue - Yp - Yd *)
	IF 	( bIsIPart = TRUE ) 
	THEN	(* I-part exists independent from the D-part *)
		(* Normal:  fYI = fYI_1 + fDi * (fE + fE_1) *)
		fYD 											:= fYD_1	:= 0.0;								
		fYI												:= fYI_1	:= MemSyncValue - fYP - fYD;	
		fY												:= MemSyncValue;
	ELSIF ( bIsDPart = TRUE ) 
	THEN	(* no I-part available, only D-part exits *)
		(* Normal:  fYD = fCd * fYD_1 + fDd * (fE - fE_1) *)
		(* fYD := fYD_1 := (fSyncValue - fYP - fYI) / fCd;*)(* 1) pre-calculation for the next cycle; fYI must be zero because there exists no I-part *)
		fYD												:= fYD_1	:= (MemSyncValue - fYP - fYI);		(* 2) fYI must be zero because there exists no I-part *)
		fY												:= MemSyncValue;
	END_IF                              				
	
	Synchronize											:= TRUE;
END_METHOD

END_FUNCTION_BLOCK

// ---- POUs/ControllerTools/signum.TcPOU
//LREAL Signum function
FUNCTION signum : LREAL
VAR_INPUT
	IN		:	LREAL;
END_VAR
VAR
END_VAR

IF IN = 0.0
THEN
	SIGNUM		:= 0.0;
ELSIF IN > 0.0
THEN
	SIGNUM		:= 1.0;
ELSE
	SIGNUM	 	:= -1.0;
END_IF

END_FUNCTION

// ---- POUs/DataBuffer/DoubleBuffer.TcPOU
//Double buffer FB to fill one part of buffer while the other (filled) part can be read or processed meanwhile
//Variable "ReadyToRead" signals that recorded data can be read consistent by pointer "pDataToRead" 
//After the data are processed or copied, it is needed to call the method "setReadyToReady(Status := FALSE)" and release the buffer to be used if the other half is filled 
//With setReadyToReady(Status := TRUE) you can mark the current write buffer as "ReadyToRead" on demand and accessible via "pDataToRead"  (e.g. if no more data need to be recorded)
{attribute 'enable_dynamic_creation'}
FUNCTION_BLOCK DoubleBuffer
VAR_OUTPUT CONSTANT 	
END_VAR                     								
VAR_INPUT
	Overwrite												:	BOOL ; //Overwrite buffer read buffer if not released -> setReadyToRead(FALSE)        
	SizeOfMemory											: 	UDINT := 5120;	//Total size of dynamic allocated buffer (will be splited in half)	   								
END_VAR                     								
VAR_IN_OUT                  								
END_VAR                     								
VAR_OUTPUT       
	TimeFillBuffer											: 	TIME; //Last elapsed time to fill the buffer and set ReadyToRead=TRUE
	MinTimeFillBuffer										:	TIME; //Min time to fill buffer
	MaxTimeFillBuffer										:	TIME; //Max time to fill buffer
	Full													:	BOOL; //Buffer is full
	Empty													:	BOOL := TRUE; //Buffer is empty 
	ReadyToRead												:	BOOL; //TRUE = Data are ready and can be read via "pDataToRead" to process 
	pDataToRead												:	POINTER TO BYTE; //Pointer to recorded data/filled buffer	
	SizeOfDataToRead										:	UDINT; //Count of bytes in filled buffer ready to ready 
{attribute 'displaymode':='hex'}
	hr														:	HRESULT; //Last result of method call
END_VAR                     								
VAR            
//local ************************************************************************************
	Interlock												:	BOOL; //Task interlock
	Buffer2Active											:	BOOL; //Indicates active buffer pointer 
	pBuffer1												: 	POINTER TO BYTE; //Pointer to start of allocated memory
	pBuffer2												: 	POINTER TO BYTE; //Pointer to second half of allocated memory
	StartTimeFillBuffer										:	TIME;
	
	MemSizeOfAllocatedMemory								: 	UDINT; //Total size of allocated memory
	MemSizeOfBuffer											: 	UDINT; //Size of split buffer
	MemSizeOfWriteBuffer									:	UDINT; //Actual size of recorded data


//trigger *********************************************************************************

//timer ***********************************************************************************

//instances ***********************************************************************************             								

//Dummys ****************************************************************************************

END_VAR

METHOD PUBLIC addData : HRESULT //Add data to write buffer and sets "ReadyToRead" if buffer is filled and data can be read to process 
VAR_INPUT
	pData													:	POINTER TO BYTE;
	SizeofData												:	UDINT;
END_VAR

IF pData <> 0 
THEN		
	//Allocate Memory to buffer messages
	IF pBuffer1 = 0
		OR SizeOfMemory > MemSizeOfAllocatedMemory 
	THEN //Allocate full memory with first entry 		
		IF NOT Allocate(SizeOfMemory)
		THEN
			addData := hr										:= E_HRESULTADSERR.NOMEMORY;
			RETURN;														
		END_IF					
	END_IF	

	IF MemSizeOfWriteBuffer = 0 THEN StartTimeFillBuffer := TIME(); END_IF
	
	//Change buffer if filled
	IF SizeofData + MemSizeOfWriteBuffer >= MemSizeOfBuffer
	THEN
		IF setReadyToRead(TRUE) <> S_OK
		THEN
			addData 											:= hr;
			RETURN;
		END_IF
	ELSE
		Full													:= FALSE;
		Empty													:= FALSE;
	END_IF
			
	//Copy data to buffer
	MEMCPY(SEL(Buffer2Active, pBuffer1, pBuffer2) + MemSizeOfWriteBuffer, pData, SizeofData);
	MemSizeOfWriteBuffer										:= MemSizeOfWriteBuffer + SizeofData;
	
	addData := hr												:= S_OK;
ELSE
	addData := hr												:= E_HRESULTADSERR.INVALIDPARM;
END_IF
END_METHOD

METHOD PUBLIC addString : HRESULT //Add string to write buffer and sets "ReadyToRead" if buffer is filled and data can be read to process 
VAR_INPUT
	Data													:	T_MAXSTRING;
END_VAR
addString := hr := addData(ADR(Data),TO_UDINT(LEN(Data)));
END_METHOD

METHOD PROTECTED FINAL allocate : BOOL //allocte buffer memory form router pool
VAR_INPUT
	SizeOfBuffer											:	UDINT;
END_VAR
VAR
	pDummy													:	POINTER TO BYTE;	
End_Var
IF SizeOfBuffer	= 0
THEN
	Allocate												:= FALSE;
	
ELSIF pBuffer1 = 0
THEN
	MemSizeOfAllocatedMemory								:= SizeOfBuffer;
	pBuffer1												:= __NEW(BYTE,MemSizeOfAllocatedMemory );
	MemSizeOfBuffer											:= MemSizeOfAllocatedMemory / 2;
	pBuffer2												:= pBuffer1 + MemSizeOfBuffer; 
	Buffer2Active											:= FALSE;
	MemSizeOfWriteBuffer									:= 0;
	
	IF PARAM.ENABLE_DEBUG_MSG_DYNAMIC_MEM_ALLOCATION
	THEN
		AdsLogHint('EngineeringToolbox | FB DoubleBuffer | An instance allocated %s bytes from the dynamic memory of the ADS router memory pool', TO_STRING(MemSizeOfAllocatedMemory));
	END_IF	
	Allocate												:= TRUE;
ELSIF SizeOfBuffer > MemSizeOfBuffer 
THEN //Since increased, allocate new memory
	
	pDummy													:= __NEW(BYTE, SizeOfBuffer); 

	IF SizeOfBuffer > MemSizeOfAllocatedMemory
	THEN //Size increased rescue data from old memory
		IF Buffer2Active
		THEN
			MEMCPY(pDummy,pBuffer2, MemSizeOfBuffer);
		ELSE
			MEMCPY(pDummy,pBuffer1, MemSizeOfBuffer);	
		END_IF
	END_IF

	__DELETE(pBuffer1);  //Delete reference to old memory
	
	MemSizeOfAllocatedMemory								:= SizeOfBuffer;
	pBuffer1												:= pDummy; //Take over new pointer to new memory
	Buffer2Active											:= FALSE;
	MemSizeOfBuffer											:= MemSizeOfAllocatedMemory / 2;
	pBuffer2												:= pBuffer1 + MemSizeOfBuffer; 
	MemSizeOfWriteBuffer										:= 0;
	
	IF PARAM.ENABLE_DEBUG_MSG_DYNAMIC_MEM_ALLOCATION
	THEN
		AdsLogWarn('EngineeringToolbox | FB DoubleBuffer | Value of "SizeOfMemory" increased and an instance has an additional %s bytes allocated from the dynamic memory of the ADS router memory pool', TO_STRING(MemSizeOfAllocatedMemory));
	END_IF
	
	Allocate												:= TRUE;
	
ELSE //Size decreased
	Allocate												:= TRUE;
END_IF
END_METHOD

METHOD PUBLIC copyData : HRESULT //Copy data from buffer (pDataToRead) into destination and reset "ReadyToReady" back to false if succeful executed 
VAR_INPUT
	pDest													:	POINTER TO BYTE; 
	SizeOfDest												:	UDINT; //Size of destination/data to copy
END_VAR
IF pDest <> 0 AND SizeOfDest > 0
	AND pDataToRead <> 0 
THEN
	MEMCPY(pDest, pDataToRead, MIN(SizeOfDest,SizeOfDataToRead));										
	hr		 												:= setReadyToRead(FALSE);	
	
ELSE
	IF pDataToRead = 0
	THEN
		hr													:= E_HRESULTADSERR.NOTREADY;
	ELSIF pDest = 0 
	THEN 
		hr													:= E_HRESULTADSERR.INVALIDPARM;
	ELSIF SizeOfDest = 0
	THEN
		hr													:= E_HRESULTADSERR.INVALIDPARM;	
	END_IF
END_IF
copyData													:= hr;
END_METHOD

METHOD FB_exit : BOOL
VAR_INPUT
	bInCopyCode : BOOL; // if TRUE, the exit method is called for exiting an instance that is copied afterwards (online change).
END_VAR
IF NOT bInCopyCode AND pBuffer1 <> 0
THEN //Release memory in case the PLC stopps
	__DELETE(pBuffer1);
END_IF
END_METHOD

{attribute 'monitoring' := 'call'}
PROPERTY PUBLIC fillLevel : INT //Buffer fill level 100% if both parts of buffer are filled
GET
IF MemSizeOfBuffer <> 0
THEN
	fillLevel												:= 	TO_INT((50.0 / TO_LREAL(MemSizeOfBuffer)) * TO_LREAL(MemSizeOfWriteBuffer))
																+ SEL(ReadyToRead, 0, TO_INT((50.0 / TO_LREAL(MemSizeOfBuffer)) * TO_LREAL(SizeOfDataToRead)));
ELSE
	fillLevel												:= 0;
END_IF
END_GET
END_PROPERTY

//Reset buffer 
METHOD PUBLIC reset : BOOL //TRUE if method is finnished
VAR_INPUT
END_VAR
TimeFillBuffer												:= T#0MS;
MinTimeFillBuffer											:= T#0MS;
MaxTimeFillBuffer											:= T#0MS;
Full														:= FALSE; //Buffer is full
Empty														:= TRUE; //Buffer is empty 
ReadyToRead													:= FALSE;
SizeOfDataToRead											:= 0;
hr															:= S_OK;
MemSizeOfWriteBuffer										:= 0;
reset														:= TRUE;
END_METHOD

METHOD PUBLIC setReadyToRead : HRESULT //Status = FALSE to reset "ReadyToRead" and unlock buffer / Status = TRUE to mark current write buffer as filled and "ReadyToRead", accessible via "pDataToRead"
VAR_INPUT
	Status								:	BOOL; //FALSE to reset "ReadyToRead" or TRUE to set "ReadyToRead" and swap buffer 
END_VAR
IF TestAndSet(Interlock)
THEN
	IF NOT Status
	THEN
		ReadyToRead									:= FALSE;
		Full										:= FALSE;
		Empty										:= MemSizeOfWriteBuffer = 0;
		hr											:= S_OK;
	ELSIF Overwrite 
		OR NOT ReadyToRead
	THEN //Set ready to ready and swap buffer
		hr											:= SEL(swapBuffer(), E_HRESULTADSERR.ABORTED ,S_OK);
		TimeFillBuffer								:= TIME() - StartTimeFillBuffer;
		IF MinTimeFillBuffer = T#0MS THEN MinTimeFillBuffer := TimeFillBuffer; ELSE MinTimeFillBuffer := MIN(TimeFillBuffer,MinTimeFillBuffer); END_IF	
		MaxTimeFillBuffer							:= MAX(TimeFillBuffer,MaxTimeFillBuffer);
		StartTimeFillBuffer							:= TIME();
		ReadyToRead									:= SizeOfDataToRead > 0;
		Full										:= FALSE;
		Empty										:= NOT ReadyToRead;
	ELSE
		TimeFillBuffer								:= TIME() - StartTimeFillBuffer;
		IF MinTimeFillBuffer = T#0MS THEN MinTimeFillBuffer := TimeFillBuffer; ELSE MinTimeFillBuffer := MIN(TimeFillBuffer,MinTimeFillBuffer); END_IF
		MaxTimeFillBuffer							:= MAX(TimeFillBuffer,MaxTimeFillBuffer);
		StartTimeFillBuffer							:= TIME();		
		Full										:= TRUE;
		Empty										:= FALSE;
		hr											:= E_HRESULTADSERR.ABORTED;	
	END_IF
		
	setReadyToRead									:= hr;
	Interlock										:= FALSE;
ELSE
	setReadyToRead									:= E_HRESULTADSERR.BUSY;
END_IF
END_METHOD

METHOD PROTECTED FINAL swapBuffer : BOOL //swap write and read buffer and asign filled buffer to pDataToRead
VAR_INPUT
END_VAR
pDataToRead													:= SEL(Buffer2Active, pBuffer1, pBuffer2);
SizeOfDataToRead											:= MemSizeOfWriteBuffer;	

Buffer2Active												:= NOT Buffer2Active;	

MemSizeOfWriteBuffer										:= 0;
swapBuffer													:= TRUE;
END_METHOD

END_FUNCTION_BLOCK

// ---- POUs/Logging/adsLogHint.TcPOU
{attribute 'no_check' := ''}
//Writes a string as a hint message into the TwinCAT AMS Logger and Windows Event Log with an possible argument
//Please see Beckhoff information system "ADSLOGxxxx" for detailed information.
//Intention of this function is to use the handy ADSLOGxxxx with a predefined msgCtrlMask of "ADSLOG_MSGTYPE_STRING OR ADSLOG_MSGTYPE_HINT OR ADSLOG_MSGTYPE_LOG"
FUNCTION adsLogHint : DINT//Write hint message into ADS log windows - Return value will be error code or 0 if OK
VAR_INPUT               											
	MsgFmtStr												:	T_MaxString; ///Message text with %s as placeholder for StrArg
(*	dintArg													:	DINT; //DINT argument for message - to be replaced by %d *) 
	StrArg													:	T_MaxString; //String argument for message - to be replaced by %s
(*	realArg													:	LREAL; //LREAL argument for message - to be replaced by %f *) 
END_VAR
VAR
	msgCtrlMask												:	DWORD; (* 	ADSLOG_MSGTYPE_HINT Meldungstyp ist Hinweis.
																				ADSLOG_MSGTYPE_WARN Meldungstyp ist Warnung.  
																				ADSLOG_MSGTYPE_ERROR Meldungstyp ist Fehler.  
																				ADSLOG_MSGTYPE_LOG Meldung wird in das Logbuch geschrieben.  
																				ADSLOG_MSGTYPE_MSGBOX Meldung wird in einer Messagebox ausgegeben.  
																				ADSLOG_MSGTYPE_RESOURCE Meldung wird aus einer Ressource-Datei geholt. (wird momentan nicht  unterstützt)  
																				ADSLOG_MSGTYPE_STRING 	Meldung ist direkt angegebener String (default).  *)	
END_VAR

(* create fixed message ctrl mask **********************************)
	msgCtrlMask												:= ADSLOG_MSGTYPE_STRING OR ADSLOG_MSGTYPE_HINT OR ADSLOG_MSGTYPE_LOG;

(* write string which includes a floating-number ******************)
(*	AdsLogHint 												:= ADSLOGLREAL(msgCtrlMask, msgFmtStr, realArg); *)
	
(* write string which includes a DINT-number *******************)
(*	AdsLogHint 												:= ADSLOGDINT(msgCtrlMask, msgFmtStr, dintArg); *)

(* write string which includes an other string e.g. 'hallo: %s what's up' ***************)
	adsLogHint 												:= ADSLOGSTR(msgCtrlMask, msgFmtStr,strArg); 

(*****************************************************)

END_FUNCTION

// ---- POUs/DataBuffer/FiFo/Fifo.TcPOU
//Fifo base control template with external memory based of FifoBase
FUNCTION_BLOCK Fifo EXTENDS FifoBase
VAR_INPUT
END_VAR
VAR_OUTPUT
END_VAR
VAR
END_VAR

;

//Clear out one entry from the Fifo buffer
METHOD PUBLIC clear : BOOL //TRUE if method was successful
VAR_INPUT
	EntryNo													:	UDINT;
	pMemory													: 	POINTER TO BYTE := 0;
	SizeOfMemory											: 	UDINT := 0;
END_VAR             										
VAR                 										
END_VAR
Clear := SUPER^._Clear(EntryNo,pMemory,SizeOfMemory);
END_METHOD

//Clear out defined data set from the Fifo buffer
METHOD PUBLIC clearByDataSet : BOOL //TRUE if method was successful
VAR_INPUT
	pData													: 	POINTER TO BYTE := 0;
	SizeOfData												: 	UDINT := 0;										
	pMemory													: 	POINTER TO BYTE := 0;
	SizeOfMemory											: 	UDINT := 0;
END_VAR             										
VAR         
	i														:	DINT;        										
END_VAR
ClearByDataSet := SUPER^._ClearByDataSet(pData,SizeOfEntry,pMemory,SizeOfMemory);
END_METHOD

METHOD PUBLIC dequeue : BOOL //TRUE if method was successful
VAR_INPUT
	pData													: 	POINTER TO BYTE := 0;
	SizeOfData												: 	UDINT := 0;
	pMemory													: 	POINTER TO BYTE := 0;
	SizeOfMemory											: 	UDINT := 0;
END_VAR
Dequeue := SUPER^._Dequeue(pData,SizeOfEntry,pMemory,SizeOfMemory);
END_METHOD

METHOD PUBLIC enqueue : BOOL //TRUE if method was successful
VAR_INPUT
	pData													: 	POINTER TO BYTE := 0;
	SizeOfData												: 	UDINT := 0;
	pMemory													: 	POINTER TO BYTE := 0;
	SizeOfMemory											: 	UDINT := 0;
END_VAR
Enqueue := SUPER^._Enqueue(pData,SizeOfData,pMemory,SizeOfMemory);
END_METHOD

//Check wheter a value already exist
METHOD PUBLIC isEnqueued : uDINT //data exist in Fifo if reurn value <> 0, returns index of entry in buffer 
VAR_INPUT
	pData													: 	POINTER TO BYTE := 0;
	SizeOfData												: 	UDINT := 0;
	pMemory													: 	POINTER TO BYTE := 0;
	SizeOfMemory											: 	UDINT := 0;
END_VAR	
VAR
	i 														: 	DINT;
END_VAR
IsEnqueued := SUPER^._IsEnqueued(pData,SizeOfEntry,pMemory,SizeOfMemory);
END_METHOD

//Check wheter a value will be the next output of the buffer
METHOD PUBLIC isNextEntry : BOOL //Inputs value is the next output 
VAR_INPUT
	pData													: 	POINTER TO BYTE := 0;
	SizeOfData												: 	UDINT := 0;
	pMemory													: 	POINTER TO BYTE := 0;
	SizeOfMemory											: 	UDINT := 0;
END_VAR
VAR
END_VAR
IsNextEntry := SUPER^._IsNextEntry(pData,SizeOfEntry,pMemory,SizeOfMemory);
END_METHOD

METHOD PUBLIC readEntry : BOOL //TRUE if method was successful
VAR_INPUT
	idx														:	UDINT;
	pData													: 	POINTER TO BYTE := 0;
	SizeOfData												: 	UDINT := 0;
	pMemory													: 	POINTER TO BYTE := 0;
	SizeOfMemory											: 	UDINT := 0;
END_VAR
ReadEntry := SUPER^._ReadEntry(idx,pData,SizeOfEntry,pMemory,SizeOfMemory);
END_METHOD

//Reset complete Fifo
METHOD PUBLIC reset : BOOL //TRUE if method is finnished
VAR_INPUT
	pMemory													: 	POINTER TO BYTE := 0;
	SizeOfMemory											: 	UDINT := 0;
END_VAR
reset := SUPER^._reset(pMemory,SizeOfMemory);
END_METHOD

END_FUNCTION_BLOCK

// ---- POUs/DataBuffer/FiFo/FiFoExt.TcPOU
//FifoBase extended with dynamical memory allocation
 {attribute 'enable_dynamic_creation'}
FUNCTION_BLOCK FiFoExt EXTENDS FifoBase
VAR_OUTPUT CONSTANT
END_VAR   
VAR_INPUT
	MaxNoOfEntrys											: 	UDINT := 10;	//0 = dynamically allocation / <> 0 = pre allcoation of memory based on size of first entry (n * data size) 
END_VAR
VAR_OUTPUT
	pMemory													: 	POINTER TO BYTE := 0; //Pointer to memory	
	SizeOfMemory											: 	UDINT := 0; //According MaxNoOfEntrys and SizeOfData of first entry
END_VAR
VAR
	MemSizeAllocatedMemory									:	UDINT := 0; //Allocated memory 
	MemSizeOfData											:	UDINT;
	MemMaxNoOfEntrys										:	UDINT;
	ExtInterlock											:	BOOL;
END_VAR

;

METHOD PROTECTED FINAL allocate : BOOL
VAR_IN_OUT
	SizeOfData												:	UDINT;
END_VAR
VAR
	pDummy													:	POINTER TO BYTE;	
End_Var
IF pMemory = 0
THEN
	IF SizeOfData = 0 OR MaxNoOfEntrys = 0
	THEN
		Allocate											:= FALSE;	
	ELSE
		MemSizeOfData										:= SizeOfData;
		MemMaxNoOfEntrys									:= MaxNoOfEntrys;
		SizeOfMemory										:= MemSizeOfData * MemMaxNoOfEntrys;
		MemSizeAllocatedMemory								:= SizeOfMemory;
		pMemory												:= __NEW(BYTE,SizeOfMemory );
		
		IF PARAM.ENABLE_DEBUG_MSG_DYNAMIC_MEM_ALLOCATION
		THEN
			AdsLogHint('EngineeringToolbox | FB FifoExt | An instance allocated %s bytes from the dynamic memory of the ADS router memory pool', TO_STRING(SizeOfMemory));
		END_IF
	END_IF

ELSIF SizeOfData = MemSizeOfData AND MaxNoOfEntrys = MemMaxNoOfEntrys
THEN
	Allocate												:= TRUE;
	
ELSIF SizeOfData > MemSizeOfData OR MaxNoOfEntrys > MemMaxNoOfEntrys
THEN //Since increased, allocate new memory
	MemSizeAllocatedMemory									:= SizeOfData * MaxNoOfEntrys;
	pDummy													:= __NEW(BYTE, MemSizeAllocatedMemory); 
	
	 //Size of data still the same, copy old data to reuse
	IF MemSizeOfData = SizeOfData AND Count > 0
	THEN
		MEMCPY(pDummy,pMemory, SizeOfMemory);
	END_IF
	
	//Copy new settings to local variales
	MemSizeOfData											:= SizeOfData;
	MemMaxNoOfEntrys										:= MaxNoOfEntrys;	
	SizeOfMemory 											:= MemSizeAllocatedMemory;

	__DELETE(pMemory);  //Delete reference to old memory
	pMemory													:= pDummy; //Take over new pointer to new memory
	
	IF PARAM.ENABLE_DEBUG_MSG_DYNAMIC_MEM_ALLOCATION
	THEN
		AdsLogWarn('EngineeringToolbox | FB FifoExt | Value of "MaxNoOfEntrys" or data size increased and one instance allocated additional %s bytes from the dynamic memory of the ADS router memory pool', TO_STRING(SizeOfMemory));
	END_IF
	
	Allocate												:= TRUE;
	
ELSE //Size decreased
	IF MemSizeOfData <> SizeOfData AND Count > 0
	THEN //Size of data changed, erease memory 
		MEMSET(pMemory,0, MemSizeAllocatedMemory);
	ELSE //Size of data the same, keep current data
		;
	END_IF
	
	//Copy new settings to local variales
	MemSizeOfData											:= SizeOfData;
	MemMaxNoOfEntrys										:= MaxNoOfEntrys;
	SizeOfMemory											:= MemSizeOfData * MemMaxNoOfEntrys;
	Allocate												:= TRUE;
END_IF
END_METHOD

//Clear out one entry from the Fifo buffer
METHOD PUBLIC clear : BOOL //TRUE if method was successful
VAR_INPUT
	EntryNo													:	UDINT;
END_VAR             										
VAR                 										
END_VAR
Clear := SUPER^._Clear(EntryNo,This^.pMemory,This^.SizeOfMemory);
END_METHOD

//Clear out defined data set from the Fifo buffer
METHOD PUBLIC clearByDataSet : BOOL //TRUE if method was successful
VAR_INPUT
	pData													: 	POINTER TO BYTE := 0;				
END_VAR             										
VAR                 										
END_VAR
ClearByDataSet := SUPER^._ClearByDataSet(pData,SizeOfEntry,This^.pMemory,This^.SizeOfMemory);
END_METHOD

METHOD PUBLIC dequeue : BOOL //TRUE if method was successful
VAR_INPUT
	pData													:	POINTER TO BYTE;	
END_VAR
VAR
END_VAR
Dequeue := SUPER^._Dequeue(pData,SizeOfEntry,This^.pMemory,This^.SizeOfMemory);
END_METHOD

METHOD PUBLIC enqueue : BOOL //TRUE if method was successful
VAR_INPUT
	pData													:	POINTER TO BYTE;
	SizeOfData												:	UDINT;
END_VAR
VAR
	CopySize												:	UDINT;
	pDummy													:	POINTER TO BYTE;
END_VAR
IF TestAndSet(ExtInterlock) 
THEN	
	if Allocate(SizeOfData)
	then
		Enqueue 											:= SUPER^._Enqueue(pData,SizeOfData,THIS^.pMemory,THIS^.SizeOfMemory);
		ExtInterlock										:= FALSE;
	else
		Enqueue												:= FALSE;
	END_IF	
ELSE
	Enqueue													:= FALSE;
END_IF
END_METHOD

METHOD FB_exit : BOOL
VAR_INPUT
	bInCopyCode : BOOL; // if TRUE, the exit method is called for exiting an instance that is copied afterwards (online change).
END_VAR
IF NOT bInCopyCode AND pMemory <> 0
THEN //Release memory in case the PLC stopps
	__DELETE(pMemory);
	Full													:= FALSE;
	Empty													:= TRUE;
	Count													:= 0;
	SizeOfMemory											:= 0;
	MemSizeOfData											:= 0;
	MemSizeAllocatedMemory									:= 0;
	MemMaxNoOfEntrys										:= MaxNoOfEntrys;
END_IF
END_METHOD

//Check wheter a value already exist
METHOD PUBLIC isEnqueued : UDINT //pData entry exist in Fifo at idx as return value 
VAR_INPUT
	pData													: 	POINTER TO BYTE := 0;
END_VAR
IsEnqueued := SUPER^._IsEnqueued(pData,SizeOfEntry,This^.pMemory,This^.SizeOfMemory);
END_METHOD

//Check wheter a value will be the next output of the buffer
METHOD PUBLIC isNextEntry : BOOL //Inputs value is the next output 
VAR_INPUT
	pData													: 	POINTER TO BYTE := 0;
END_VAR
VAR
END_VAR
IsNextEntry := SUPER^._IsNextEntry(pData,SizeOfEntry,This^.pMemory,This^.SizeOfMemory);
END_METHOD

METHOD PUBLIC readEntry : BOOL //TRUE if method was successful
VAR_INPUT
	idx														:	UDINT;
	pData													: 	POINTER TO BYTE := 0;
END_VAR
ReadEntry := SUPER^._ReadEntry(idx,pData,SizeOfEntry,This^.pMemory,This^.SizeOfMemory);
END_METHOD

//Reset complete Fifo
METHOD PUBLIC reset : BOOL //TRUE if method is finnished
VAR_INPUT
END_VAR
reset				:= SUPER^._reset(This^.pMemory,This^.SizeOfMemory);
END_METHOD

END_FUNCTION_BLOCK

// ---- POUs/DataBuffer/FiFo/FiFoLRealSimple.TcPOU
//Fifo with a internal Lreal array for a simple num list implementation
FUNCTION_BLOCK FiFoLRealSimple EXTENDS FifoBase
VAR_OUTPUT CONSTANT
	MIN_BUFFER												:	DINT := 1; //Fifo buffer start index 
	MAX_BUFFER												:	DINT := PARAM.FIFO_LREAL_SIMPEL_MAX_BUFFER; //Fifo buffer end index - see library parameter to customize parameter
END_VAR   
VAR_INPUT
END_VAR
VAR_OUTPUT
	Buffer													:	ARRAY[MIN_BUFFER..MAX_BUFFER] OF LREAL; //Lreal Fifo buffer 
END_VAR
VAR
END_VAR

;

 //Clear out one entry from the Fifo buffer
METHOD PUBLIC clear : BOOL //TRUE if method was successful
VAR_INPUT
	EntryNo													:	UDINT;
END_VAR             										
VAR                 										
END_VAR
Clear := super^._Clear(EntryNo,ADR(Buffer),SIZEOF(Buffer));
END_METHOD

//Clear out defined data set from the Fifo buffer
METHOD PUBLIC clearByDataSet : BOOL //TRUE if method was successful
VAR_INPUT
	Value													:	LREAL;
END_VAR             										
VAR                 										
END_VAR
ClearByDataSet := super^._ClearByDataSet(ADR(Value),SIZEOF(Value),ADR(Buffer),SIZEOF(Buffer));
END_METHOD

METHOD PUBLIC dequeue : BOOL //TRUE if method was successful
VAR_IN_OUT
	Value													:	LREAL;	
END_VAR
VAR
END_VAR
Dequeue := SUPER^._Dequeue(ADR(Value),SIZEOF(Value),ADR(Buffer),SIZEOF(Buffer));
END_METHOD

METHOD PUBLIC enqueue : BOOL //TRUE if method was successful
VAR_INPUT
	Value													:	LREAL;
END_VAR
Enqueue := SUPER^._Enqueue(ADR(Value),SIZEOF(Value),ADR(Buffer),SIZEOF(Buffer));
END_METHOD

//Check wheter a value already exist
METHOD PUBLIC isEnqueued : uDINT //In Value exist in Fifo at idx as return value  
VAR_INPUT
	Value													:	LREAL;
END_VAR
IsEnqueued := SUPER^._IsEnqueued(ADR(Value),SIZEOF(Value),ADR(Buffer),SIZEOF(Buffer));
END_METHOD

//Check wheter a value will be the next output of the buffer
METHOD PUBLIC isNextEntry : BOOL //Inputs value is the next output 
VAR_INPUT
	Value													: LREAL;
END_VAR
VAR
END_VAR
IsNextEntry := SUPER^._IsNextEntry(ADR(Value),SIZEOF(Value),ADR(Buffer),SIZEOF(Buffer));
END_METHOD

METHOD PUBLIC readEntry : BOOL //TRUE if method was successful
VAR_INPUT
	idx														:	uDINT;
END_VAR
VAR_IN_OUT
	value													: LREAL;	
END_VAR
ReadEntry := SUPER^._ReadEntry(idx,ADR(Value),SIZEOF(Value),ADR(Buffer),SIZEOF(Buffer));
END_METHOD

//Reset complete Fifo
METHOD PUBLIC reset : BOOL //TRUE if method is finnished
VAR_INPUT
END_VAR
reset := SUPER^._reset(ADR(Buffer),SIZEOF(Buffer));
END_METHOD

END_FUNCTION_BLOCK

// ---- POUs/DataBuffer/LiFo/LiFoExt.TcPOU
//LifoBase extended with dynamical memory allocation
 {attribute 'enable_dynamic_creation'}
FUNCTION_BLOCK LiFoExt EXTENDS LiFoBase
VAR_OUTPUT CONSTANT
END_VAR   
VAR_INPUT
	MaxNoOfEntrys											: 	UDINT := 10;	//0 = dynamically allocation / <> 0 = pre allcoation of memory based on size of first entry (n * data size) 
END_VAR
VAR_OUTPUT
	pMemory													: 	POINTER TO BYTE := 0; //Pointer to memory	
	SizeOfMemory											: 	UDINT := 0; //According MaxNoOfEntrys and SizeOfData of first entry
END_VAR
VAR
	MemSizeAllocatedMemory									:	UDINT := 0; //Allocated memory 
	MemSizeOfData											:	UDINT;
	MemMaxNoOfEntrys										:	UDINT;
	ExtInterlock											:	BOOL;
END_VAR

;

METHOD PROTECTED FINAL allocate : BOOL
VAR_IN_OUT
	SizeOfData												:	UDINT;
END_VAR
VAR
	pDummy													:	POINTER TO BYTE;	
End_Var
IF pMemory = 0
THEN
	IF SizeOfData = 0 OR MaxNoOfEntrys = 0
	THEN
		Allocate											:= FALSE;	
	ELSE
		MemSizeOfData										:= SizeOfData;
		MemMaxNoOfEntrys									:= MaxNoOfEntrys;
		SizeOfMemory										:= MemSizeOfData * MemMaxNoOfEntrys;
		MemSizeAllocatedMemory								:= SizeOfMemory;
		pMemory												:= __NEW(BYTE,SizeOfMemory );
		
		IF PARAM.ENABLE_DEBUG_MSG_DYNAMIC_MEM_ALLOCATION
		THEN
			AdsLogHint('EngineeringToolbox | FB FifoExt | An instance allocated %s bytes from the dynamic memory of the ADS router memory pool', TO_STRING(SizeOfMemory));
		END_IF
	END_IF

ELSIF SizeOfData = MemSizeOfData AND MaxNoOfEntrys = MemMaxNoOfEntrys
THEN
	Allocate												:= TRUE;
	
ELSIF SizeOfData > MemSizeOfData OR MaxNoOfEntrys > MemMaxNoOfEntrys
THEN //Since increased, allocate new memory
	MemSizeAllocatedMemory									:= SizeOfData * MaxNoOfEntrys;
	pDummy													:= __NEW(BYTE, MemSizeAllocatedMemory); 
	
	 //Size of data still the same, copy old data to reuse
	IF MemSizeOfData = SizeOfData AND Count > 0
	THEN
		MEMCPY(pDummy,pMemory, SizeOfMemory);
	END_IF
	
	//Copy new settings to local variales
	MemSizeOfData											:= SizeOfData;
	MemMaxNoOfEntrys										:= MaxNoOfEntrys;	
	SizeOfMemory 											:= MemSizeAllocatedMemory;

	__DELETE(pMemory);  //Delete reference to old memory
	pMemory													:= pDummy; //Take over new pointer to new memory
	
	IF PARAM.ENABLE_DEBUG_MSG_DYNAMIC_MEM_ALLOCATION
	THEN
		AdsLogWarn('EngineeringToolbox | FB FifoExt | Value of "MaxNoOfEntrys" or data size increased and one instance allocated additional %s bytes from the dynamic memory of the ADS router memory pool', TO_STRING(SizeOfMemory));
	END_IF
	
	Allocate												:= TRUE;
	
ELSE //Size decreased
	IF MemSizeOfData <> SizeOfData AND Count > 0
	THEN //Size of data changed, erease memory 
		MEMSET(pMemory,0, MemSizeAllocatedMemory);
	ELSE //Size of data the same, keep current data
		;
	END_IF
	
	//Copy new settings to local variales
	MemSizeOfData											:= SizeOfData;
	MemMaxNoOfEntrys										:= MaxNoOfEntrys;
	SizeOfMemory											:= MemSizeOfData * MemMaxNoOfEntrys;
	Allocate												:= TRUE;
END_IF
END_METHOD

METHOD PUBLIC dequeue : BOOL //TRUE if method was successful
VAR_INPUT
	pData													:	POINTER TO BYTE;	
END_VAR
VAR
END_VAR
Dequeue := SUPER^._Dequeue(pData,SizeOfEntry,This^.pMemory,This^.SizeOfMemory);
END_METHOD

METHOD PUBLIC dequeueStream : BOOL //TRUE if method was successful
VAR_INPUT
	pData													: 	POINTER TO BYTE := 0;
	SizeOfStream											: 	UDINT := 0;
	pMemory													: 	POINTER TO BYTE := 0;
	SizeOfMemory											: 	UDINT := 0;
END_VAR
DequeueStream := SUPER^._DequeueStream(pData,SizeOfStream,pMemory,SizeOfMemory);
END_METHOD

METHOD PUBLIC enqueue : BOOL //TRUE if method was successful
VAR_INPUT
	pData													:	POINTER TO BYTE;
	SizeOfData												:	UDINT;
END_VAR
VAR
	CopySize												:	UDINT;
	pDummy													:	POINTER TO BYTE;
END_VAR
IF TestAndSet(ExtInterlock) 
THEN	
	if Allocate(SizeOfData)
	then
		Enqueue 											:= SUPER^._Enqueue(pData,SizeOfData,THIS^.pMemory,THIS^.SizeOfMemory);
		ExtInterlock										:= FALSE;
	else
		Enqueue												:= FALSE;
	END_IF	
ELSE
	Enqueue													:= FALSE;
END_IF
END_METHOD

METHOD PUBLIC enqueueStream : BOOL //TRUE if method was successful
VAR_INPUT
	pData													: 	POINTER TO BYTE := 0;
	SizeOfData												: 	UDINT := 0;
	SizeOfStream											: 	UDINT := 0;
	pMemory													: 	POINTER TO BYTE := 0;
	SizeOfMemory											: 	UDINT := 0;
END_VAR
EnqueueStream := SUPER^._EnqueueStream(pData,SizeOfData, SizeOfStream,pMemory,SizeOfMemory);
END_METHOD

METHOD FB_exit : BOOL
VAR_INPUT
	bInCopyCode : BOOL; // if TRUE, the exit method is called for exiting an instance that is copied afterwards (online change).
END_VAR
IF NOT bInCopyCode AND pMemory <> 0
THEN //Release memory in case the PLC stopps
	__DELETE(pMemory);
	Full													:= FALSE;
	Empty													:= TRUE;
	Count													:= 0;
	SizeOfMemory											:= 0;
	MemSizeOfData											:= 0;
	MemSizeAllocatedMemory									:= 0;
	MemMaxNoOfEntrys										:= MaxNoOfEntrys;
END_IF
END_METHOD

//Check wheter a value already exist
METHOD PUBLIC isEnqueued : UDINT //pData entry exist in Fifo at idx as return value 
VAR_INPUT
	pData													: 	POINTER TO BYTE := 0;
END_VAR
IsEnqueued := SUPER^._IsEnqueued(pData,SizeOfEntry,This^.pMemory,This^.SizeOfMemory);
END_METHOD

//Check wheter a value will be the next output of the buffer
METHOD PUBLIC isNextEntry : BOOL //Inputs value is the next output 
VAR_INPUT
	pData													: 	POINTER TO BYTE := 0;
END_VAR
VAR
END_VAR
IsNextEntry := SUPER^._IsNextEntry(pData,SizeOfEntry,This^.pMemory,This^.SizeOfMemory);
END_METHOD

METHOD PUBLIC readEntry : BOOL //TRUE if method was successful
VAR_INPUT
	idx														:	UDINT;
	pData													: 	POINTER TO BYTE := 0;
END_VAR
ReadEntry := SUPER^._ReadEntry(idx,pData,SizeOfEntry,This^.pMemory,This^.SizeOfMemory);
END_METHOD

//Reset complete Fifo
METHOD PUBLIC reset : BOOL //TRUE if method is finnished
VAR_INPUT
END_VAR
reset				:= SUPER^._reset(This^.pMemory,This^.SizeOfMemory);
END_METHOD

END_FUNCTION_BLOCK

// ---- POUs/DataBuffer/Quicksort.TcPOU
// this funktionblock sorts an array of struct by an contained element with quicksort routine
// Udpate: compare with static PivotElement
// Find Explanation under https://www.youtube.com/watch?v=eNUM23f6g-s&ab_channel=Studyflix
{attribute 'enable_dynamic_creation'}
FUNCTION_BLOCK Quicksort
VAR CONSTANT
	MAX_STRING_LENGTH										:	INT := PARAM.QUICKSORT_MAX_STRING_LENGTH;
	MAX_WSTRING_LENGTH										:	INT := PARAM.QUICKSORT_MAX_WSTRING_LENGTH;
END_VAR
VAR_INPUT
	SortInverse												:	BOOL := FALSE;//inverses order of content
	IgnoreBlank												:	BOOL := FALSE;//sort blank characters at last			
END_VAR
VAR_OUTPUT
END_VAR
VAR
	pElement_Tmp											:	POINTER TO BYTE;		// Copy Pointer 3 - allocated memory
	MemSizeOfStruct											:	UDINT;
END_VAR

;

METHOD PROTECTED FINAL allocate : BOOL
VAR_INPUT
	SizeOfStruct											: 	UDINT;	
END_VAR
IF SizeOfStruct = 0
THEN
	allocate												:= FALSE;
ELSIF pElement_Tmp = 0 
THEN
	pElement_Tmp											:= __NEW(BYTE, SizeOfStruct);
	MemSizeOfStruct											:= SizeOfStruct;
	IF TRUE
	THEN
		AdsLogHint('EngineeringToolbox | FB Quicksort | An instance allocated %s bytes from the dynamic memory of the ADS router memory pool', TO_STRING(MemSizeOfStruct));
	END_IF
	Allocate												:= TRUE;
ELSIF SizeOfStruct > MemSizeOfStruct
THEN
	__DELETE(pElement_Tmp);	
	pElement_Tmp											:= __NEW(BYTE, SizeOfStruct);
	MemSizeOfStruct											:= SizeOfStruct;
		IF TRUE
	THEN
		AdsLogWarn('EngineeringToolbox | FB Quicksort | SizeOfStruct increased and an instance has an additional %s bytes allocated from the dynamic memory of the ADS router memory pool', TO_STRING(MemSizeOfStruct));
	END_IF
	Allocate												:= TRUE;
ELSE
	Allocate												:= TRUE;	
END_IF
END_METHOD

METHOD byDINT : BOOL // returns true if sort ends successfully 
VAR_INPUT
	pData													: 	POINTER TO BYTE := 0;	// ADR(Array) 	
	SizeOfData												: 	UDINT := 0;				// SIZEOF(Array)
	pCompareElement											: 	POINTER TO BYTE := 0;	// ADR(Array[1].DINT)		
	SizeOfStruct											: 	UDINT := 0;				// SIZEOF(Array[1]) 	
END_VAR                                                 
VAR        
	pPivotElement											: 	POINTER TO DINT;		// Pivot value
	PivotElement											: 	DINT;					// Pivot value as DINT	
	pCmpElement												:	POINTER TO DINT;		// compare value
	                                					                            	
	endMainLoop												:	BOOL;					// End of main loop reached
	endSubLoop												:	BOOL;					// End of sub loop reached                                              
	ElementCount											:	DINT;					// No of array elements
	stackCount,left,right,i,j								:	DINT;					// running variables 	
	stack													:	ARRAY[1..32] OF UDINT;	// stack size 32 => ~1 Mio elements *)	
	                                					
	pElement_1												:	POINTER TO BYTE;		// Copy Pointer 1		
	pElement_2												:	POINTER TO BYTE;		// Copy Pointer 2

END_VAR
// ends with true in case of no error	                                    					 					
IF SizeOfStruct = 0 OR SizeOfData = 0
	OR pData = 0 OR pCompareElement = 0
THEN               					                                   					
	byDINT													:= FALSE;
	RETURN;   
ELSE
	byDINT													:= TRUE;                          					
END_IF                                  					
          
// calculate no. of Elements                                
ElementCount												:= TO_DINT(SizeOfData / SizeOfStruct);   		
			
// Quicksort                            					
// initial value of array size          					
left 														:= 1;				// first element
right 														:= ElementCount;	// last element 
stackCount 													:= 1;				// running variable 
                                        	
WHILE NOT endMainLoop DO							
	IF left < right THEN                	
		pPivotElement										:= pCompareElement + (SizeOfStruct * TO_UDINT(SHR(right+left,1)));
		PivotElement										:= pPivotElement^;
		i 													:= left -1;
		j 													:= right +1;
		endSubLoop 											:= FALSE;
		REPEAT
			IF SortInverse
			THEN	// sort descending	
				REPEAT	
					i 										:= i+1;	
					pCmpElement								:= pCompareElement + (SizeOfStruct * TO_UDINT(i-1));
				UNTIL (pCmpElement^ <= PivotElement) OR NOT (i < right)	END_REPEAT	
				REPEAT	
					j 										:= j-1;	
					pCmpElement								:= pCompareElement + (SizeOfStruct * TO_UDINT(j-1));
				UNTIL (pCmpElement^ >= PivotElement) OR NOT (j > left)	END_REPEAT		
			ELSE	// sort ascending
				REPEAT	
					i 										:= i+1;
					pCmpElement								:= pCompareElement + (SizeOfStruct * TO_UDINT(i-1));
				UNTIL (pCmpElement^ >= PivotElement)	OR NOT (i < right)	END_REPEAT;				
				REPEAT	
					j 										:= j-1;	
					pCmpElement								:= pCompareElement + (SizeOfStruct * TO_UDINT(j-1));
				UNTIL (pCmpElement^ <= PivotElement) OR NOT (j > left)	END_REPEAT;
			END_IF
			IF i >= j THEN
				endSubLoop									:= TRUE;
			ELSE                    					
				Allocate( SizeOfStruct);
				pElement_1									:= pData + (SizeOfStruct * TO_UDINT(j-1));
				pElement_2									:= pData + (SizeOfStruct * TO_UDINT(i-1));
				
				IF pElement_Tmp = 0 
					OR_ELSE MEMCPY(pElement_Tmp, pElement_1,	SizeOfStruct) = 0
					OR_ELSE MEMCPY(pElement_1,	pElement_2,		SizeOfStruct) = 0
					OR_ELSE MEMCPY(pElement_2,	pElement_Tmp,	SizeOfStruct) = 0
				THEN
					byDINT									:= FALSE;
					RETURN;	
				END_IF
	
			END_IF
		UNTIL endSubLoop END_REPEAT;		
		stack[stackCount] 									:= TO_UDINT(right); 	// save right in stack			
		IF stackCount < 32              					
		THEN                            					
			stackCount 										:= stackCount +1;
		ELSE															// Error stack Limit    
			endMainLoop 									:= TRUE;
			byDINT											:= FALSE;			
		END_IF                          					
		right 												:= MAX(left, i-1);
	ELSE                                
		IF stackCount = 1 THEN          
			endMainLoop 									:= TRUE;
		ELSE                            					
			left 											:= right+1;       
			stackCount 										:= stackCount -1;	// load from stack
			right											:= TO_DINT(stack[stackCount]);
		END_IF
	END_IF
END_WHILE
END_METHOD

METHOD byDINT_Bubble : BOOL // returns true if sort ends successfully 
VAR_INPUT	
	pData													:	POINTER TO BYTE;// ADR(Array) 			
	SizeOfData												:	UDINT;			// SIZEOF(Array)
	pCompareElement											:	POINTER TO BYTE;// ADR(Array[1].DINT)		
	SizeOfStruct											:	UDINT;			// SIZEOF(Array[1]) 			
END_VAR                                 					                
VAR                                     					                
	Run  													:	DINT;			// main loop
  	Index													:	DINT;			// sub loop 	
	ElementCount											:	DINT;			
	                                    					
	CompareElement_1										:	DINT;					
	CompareElement_2										:	DINT;					
	pCompareElement_1										:	POINTER TO DINT;		
	pCompareElement_2										:	POINTER TO DINT;
		                                					                        
	pElement_1												:	POINTER TO BYTE;		
	pElement_2												:	POINTER TO BYTE;		
END_VAR
// ends with true in case of no error	                                    					 					
IF SizeOfStruct = 0 OR SizeOfData = 0
	OR pData = 0 OR pCompareElement = 0
THEN               					                                   					
	byDINT_Bubble											:= FALSE;
	RETURN;   
ELSE
	byDINT_Bubble											:= TRUE;                          					
END_IF    

// Bubblesort Routine
// Code saving 
	
// calculate no. of Elements                                
ElementCount												:= TO_DINT(SizeOfData / SizeOfStruct);  

// bubblesort 
FOR Run := 1 TO TO_DINT(ElementCount) - 1 DO
    FOR Index := ElementCount - 1 TO Run BY -1 DO
		// get element x for compare 
		pCompareElement_1				:=	pCompareElement + (SizeOfStruct * TO_UDINT(Index));
		CompareElement_1				:=	pCompareElement_1^;
		// get element x-1 for compare 
		pCompareElement_2				:=	pCompareElement + (SizeOfStruct * TO_UDINT(Index-1));
		CompareElement_2 				:=	pCompareElement_2^;
		// switch by useing temporary memory 
		IF ((	CompareElement_1 < CompareElement_2) AND NOT SortInverse)
			OR((CompareElement_1 > CompareElement_2) AND SortInverse)
		THEN
			// get pointer for MEMCPY 
			Allocate(SizeOfStruct);
			pElement_1					:= pData + SizeOfStruct * TO_UDINT(Index);
			pElement_2					:= pData + SizeOfStruct * TO_UDINT(Index-1);
			
	
			IF pElement_Tmp = 0 
				OR_ELSE MEMCPY(pElement_Tmp, pElement_1,	SizeOfStruct) = 0
				OR_ELSE MEMCPY(pElement_1,	pElement_2,		SizeOfStruct) = 0
				OR_ELSE MEMCPY(pElement_2,	pElement_Tmp,	SizeOfStruct) = 0
			THEN
				byDINT_Bubble		:= FALSE;
				EXIT;												
			END_IF

      END_IF
	END_FOR
END_FOR
END_METHOD

METHOD byINT : BOOL // returns true if sort ends successfully 
VAR_INPUT
	pData													: 	POINTER TO BYTE := 0;	// ADR(Array) 	
	SizeOfData												: 	UDINT := 0;				// SIZEOF(Array)
	pCompareElement											: 	POINTER TO BYTE := 0;	// ADR(Array[1].INT)		
	SizeOfStruct											: 	UDINT := 0;				// SIZEOF(Array[1]) 	
END_VAR                                                 
VAR        
	pPivotElement											: 	POINTER TO INT;			// Pivot value
	PivotElement											: 	INT;					// Pivot value as INT	
	pCmpElement												:	POINTER TO INT;			// compare value
	                                					                            	
	endMainLoop												:	BOOL;					// End of main loop reached
	endSubLoop												:	BOOL;					// End of sub loop reached                                              
	ElementCount											:	DINT;					// No of array elements
	stackCount,left,right,i,j								:	DINT;					// running variables 	
	stack													:	ARRAY[1..32] OF UDINT;	// stack size 32 => ~1 Mio elements *)	
	                                					
	pElement_1												:	POINTER TO BYTE;		// Copy Pointer 1		
	pElement_2												:	POINTER TO BYTE;		// Copy Pointer 2
END_VAR
// ends with true in case of no error	                                    					 					
IF SizeOfStruct = 0 OR SizeOfData = 0
	OR pData = 0 OR pCompareElement = 0
THEN               					                                   					
	byINT													:= FALSE;
	RETURN;   
ELSE
	byINT													:= TRUE;                          					
END_IF                                    					
        
// calculate no. of Elements                                
ElementCount												:= TO_DINT(SizeOfData / SizeOfStruct);   
                                					
// Quicksort                            					
// initial value of array size          					
left 														:= 1;				// first element
right 														:= ElementCount;	// last element 
stackCount 													:= 1;				// running variable 
                                        	
WHILE NOT endMainLoop DO							
	IF left < right THEN                	
		pPivotElement										:= pCompareElement + (SizeOfStruct * TO_UDINT(SHR(right+left,1)));
		PivotElement										:= pPivotElement^;
		i 													:= left -1;
		j 													:= right +1;
		endSubLoop 											:= FALSE;
		REPEAT
			IF SortInverse
			THEN	// sort descending	
				REPEAT	
					i 										:= i+1;	
					pCmpElement								:= pCompareElement + (SizeOfStruct * TO_UDINT(i-1));
				UNTIL (pCmpElement^ <= PivotElement) OR NOT (i < right)	END_REPEAT	
				REPEAT	
					j 										:= j-1;	
					pCmpElement								:= pCompareElement + (SizeOfStruct * TO_UDINT(j-1));
				UNTIL (pCmpElement^ >= PivotElement) OR NOT (j > left)	END_REPEAT		
			ELSE	// sort ascending
				REPEAT	
					i 										:= i+1;
					pCmpElement								:= pCompareElement + (SizeOfStruct * TO_UDINT(i-1));
				UNTIL (pCmpElement^ >= PivotElement)	OR NOT (i < right)	END_REPEAT;				
				REPEAT	
					j 										:= j-1;	
					pCmpElement								:= pCompareElement + (SizeOfStruct * TO_UDINT(j-1));
				UNTIL (pCmpElement^ <= PivotElement) OR NOT (j > left)	END_REPEAT;
			END_IF
			IF i >= j THEN
				endSubLoop									:= TRUE;
			ELSE                    					
				Allocate(SizeOfStruct);
				pElement_1									:= pData + (SizeOfStruct * TO_UDINT(j-1));
				pElement_2									:= pData + (SizeOfStruct * TO_UDINT(i-1));
				
				IF pElement_Tmp = 0 
					OR_ELSE MEMCPY(pElement_Tmp, pElement_1,	SizeOfStruct) = 0
					OR_ELSE MEMCPY(pElement_1,	pElement_2,		SizeOfStruct) = 0
					OR_ELSE MEMCPY(pElement_2,	pElement_Tmp,	SizeOfStruct) = 0
				THEN
					byINT									:= FALSE;
					RETURN;	
				END_IF
	
			END_IF
		UNTIL endSubLoop END_REPEAT;		
		stack[stackCount] 									:= TO_UDINT(right); 	// save right in stack			
		IF stackCount < 32              					
		THEN                            					
			stackCount 										:= stackCount +1;
		ELSE															// Error stack Limit    
			endMainLoop 									:= TRUE;
			byINT											:= FALSE;			
		END_IF                          					
		right 												:= MAX(left, i-1);
	ELSE                                
		IF stackCount = 1 THEN          
			endMainLoop 									:= TRUE;
		ELSE                            					
			left 											:= right+1;       
			stackCount 										:= stackCount -1;	// load from stack
			right											:= TO_DINT(stack[stackCount]);
		END_IF
	END_IF
END_WHILE
END_METHOD

METHOD byLREAL : BOOL // returns true if sort ends successfully 
VAR_INPUT
	pData													: 	POINTER TO BYTE := 0;	// ADR(Array) 	
	SizeOfData												: 	UDINT := 0;				// SIZEOF(Array)
	pCompareElement											: 	POINTER TO BYTE := 0;	// ADR(Array[1].LREAL)		
	SizeOfStruct											: 	UDINT := 0;				// SIZEOF(Array[1]) 	
END_VAR                                                 
VAR        
	pPivotElement											: 	POINTER TO LREAL;		// Pivot value	
	PivotElement											: 	LREAL;					// Pivot value as LREAL
	pCmpElement												:	POINTER TO LREAL;		// compare value
	                                					                            	
	endMainLoop												:	BOOL;					// End of main loop reached
	endSubLoop												:	BOOL;					// End of sub loop reached                                              
	ElementCount											:	DINT;					// No of array elements
	stackCount,left,right,i,j								:	DINT;					// running variables 	
	stack													:	ARRAY[1..32] OF UDINT;	// stack size 32 => ~1 Mio elements *)	
	                                					
	pElement_1												:	POINTER TO BYTE;		// Copy Pointer 1		
	pElement_2												:	POINTER TO BYTE;		// Copy Pointer 2
	
END_VAR
// ends with true in case of no error	                                    					 					
IF SizeOfStruct = 0 OR SizeOfData = 0
	OR pData = 0 OR pCompareElement = 0
THEN               					                                   					
	byLREAL													:= FALSE;
	RETURN;   
ELSE
	byLREAL													:= TRUE;                          					
END_IF                                 					
            
// calculate no. of Elements                                
ElementCount												:= TO_DINT(SizeOfData / SizeOfStruct);   
                            					
// Quicksort                            					
// initial value of array size          					
left 														:= 1;				// first element
right 														:= ElementCount;	// last element 
stackCount 													:= 1;				// running variable 
                                        	
WHILE NOT endMainLoop DO							
	IF left < right THEN                	
		pPivotElement										:= pCompareElement + (SizeOfStruct * TO_UDINT(SHR(right+left,1))); // divide by 2
		PivotElement										:= pPivotElement^;
		i 													:= left -1;
		j 													:= right +1;
		endSubLoop 											:= FALSE;
		REPEAT
			IF SortInverse
			THEN	// sort descending	
				REPEAT	
					i 										:= i+1;	
					pCmpElement								:= pCompareElement + (SizeOfStruct * TO_UDINT(i-1));
				UNTIL (pCmpElement^ <= PivotElement) OR NOT (i < right)	END_REPEAT	
				REPEAT	
					j 										:= j-1;	
					pCmpElement								:= pCompareElement + (SizeOfStruct * TO_UDINT(j-1));
				UNTIL (pCmpElement^ >= PivotElement) OR NOT (j > left)	END_REPEAT		
			ELSE	// sort ascending
				REPEAT	
					i 										:= i+1;
					pCmpElement								:= pCompareElement + (SizeOfStruct * TO_UDINT(i-1));
				UNTIL (pCmpElement^ >= PivotElement)	OR NOT (i < right)	END_REPEAT;				
				REPEAT	
					j 										:= j-1;	
					pCmpElement								:= pCompareElement + (SizeOfStruct * TO_UDINT(j-1));
				UNTIL (pCmpElement^ <= PivotElement) OR NOT (j > left)	END_REPEAT;
			END_IF
			IF i >= j THEN
				endSubLoop									:= TRUE;
			ELSE                    					
				Allocate(SizeOfStruct);
				pElement_1									:= pData + (SizeOfStruct * TO_UDINT(j-1));
				pElement_2									:= pData + (SizeOfStruct * TO_UDINT(i-1));
				
				IF pElement_Tmp = 0 
					OR_ELSE MEMCPY(pElement_Tmp, pElement_1,	SizeOfStruct) = 0
					OR_ELSE MEMCPY(pElement_1,	pElement_2,		SizeOfStruct) = 0
					OR_ELSE MEMCPY(pElement_2,	pElement_Tmp,	SizeOfStruct) = 0
				THEN
					byLREAL									:= FALSE;
					RETURN;	
				END_IF

			END_IF
		UNTIL endSubLoop END_REPEAT;		
		stack[stackCount] 									:= TO_UDINT(right); 	// save right in stack			
		IF stackCount < 32              					
		THEN                            					
			stackCount 										:= stackCount +1;
		ELSE															// Error stack Limit    
			endMainLoop 									:= TRUE;
			byLREAL											:= FALSE;			
		END_IF                          					
		right 												:= MAX(left, i-1);
	ELSE                                
		IF stackCount = 1 THEN          
			endMainLoop 									:= TRUE;
		ELSE                            					
			left 											:= right+1;       
			stackCount 										:= stackCount -1;	// load from stack
			right											:= TO_DINT(stack[stackCount]);
		END_IF
	END_IF
END_WHILE
END_METHOD

METHOD byLTIME : BOOL // returns true if sort ends successfully 
VAR_INPUT
	pData													: 	POINTER TO BYTE := 0;	// ADR(Array) 	
	SizeOfData												: 	UDINT := 0;				// SIZEOF(Array)
	pCompareElement											: 	POINTER TO BYTE := 0;	// ADR(Array[1].LTIME)		
	SizeOfStruct											: 	UDINT := 0;				// SIZEOF(Array[1]) 	
END_VAR                                                 
VAR        
	pPivotElement											: 	POINTER TO LTIME;		// Pivot value	
	PivotElement											: 	LTIME;					// Pivot value as LTIME	
	pCmpElement												:	POINTER TO LTIME;		// compare value
	                                					                            	
	endMainLoop												:	BOOL;					// End of main loop reached
	endSubLoop												:	BOOL;					// End of sub loop reached                                              
	ElementCount											:	DINT;					// No of array elements
	stackCount,left,right,i,j								:	DINT;					// running variables 	
	stack													:	ARRAY[1..32] OF UDINT;	// stack size 32 => ~1 Mio elements *)	
	                                					
	pElement_1												:	POINTER TO BYTE;		// Copy Pointer 1		
	pElement_2												:	POINTER TO BYTE;		// Copy Pointer 2
END_VAR
// ends with true in case of no error	                                    					 					
IF SizeOfStruct = 0 OR SizeOfData = 0
	OR pData = 0 OR pCompareElement = 0
THEN               					                                   					
	byLTIME													:= FALSE;
	RETURN;   
ELSE
	byLTIME													:= TRUE;                          					
END_IF                                    					
             
// calculate no. of Elements                                
ElementCount												:= TO_DINT(SizeOfData / SizeOfStruct);   
                           					
// Quicksort                            					
// initial value of array size          					
left 														:= 1;				// first element
right 														:= ElementCount;	// last element 
stackCount 													:= 1;				// running variable 
                                        	
WHILE NOT endMainLoop DO							
	IF left < right THEN                	
		pPivotElement										:= pCompareElement + (SizeOfStruct * TO_UDINT(SHR(right+left,1)));
		PivotElement										:= pPivotElement^;
		i 													:= left -1;
		j 													:= right +1;
		endSubLoop 											:= FALSE;
		REPEAT
			IF SortInverse
			THEN	// sort descending	
				REPEAT	
					i 										:= i+1;	
					pCmpElement								:= pCompareElement + (SizeOfStruct * TO_UDINT(i-1));
				UNTIL (pCmpElement^ <= PivotElement) OR NOT (i < right)	END_REPEAT	
				REPEAT	
					j 										:= j-1;	
					pCmpElement								:= pCompareElement + (SizeOfStruct * TO_UDINT(j-1));
				UNTIL (pCmpElement^ >= PivotElement) OR NOT (j > left)	END_REPEAT		
			ELSE	// sort ascending
				REPEAT	
					i 										:= i+1;
					pCmpElement								:= pCompareElement + (SizeOfStruct * TO_UDINT(i-1));
				UNTIL (pCmpElement^ >= PivotElement)	OR NOT (i < right)	END_REPEAT;				
				REPEAT	
					j 										:= j-1;	
					pCmpElement								:= pCompareElement + (SizeOfStruct * TO_UDINT(j-1));
				UNTIL (pCmpElement^ <= PivotElement) OR NOT (j > left)	END_REPEAT;
			END_IF
			IF i >= j THEN
				endSubLoop									:= TRUE;
			ELSE                    					
				Allocate(SizeOfStruct);
				pElement_1									:= pData + (SizeOfStruct * TO_UDINT(j-1));
				pElement_2									:= pData + (SizeOfStruct * TO_UDINT(i-1));
				
				IF pElement_Tmp = 0 
					OR_ELSE MEMCPY(pElement_Tmp, pElement_1,	SizeOfStruct) = 0
					OR_ELSE MEMCPY(pElement_1,	pElement_2,		SizeOfStruct) = 0
					OR_ELSE MEMCPY(pElement_2,	pElement_Tmp,	SizeOfStruct) = 0
				THEN
					byLTIME									:= FALSE;
					RETURN;	
				END_IF

			END_IF
		UNTIL endSubLoop END_REPEAT;		
		stack[stackCount] 									:= TO_UDINT(right); 	// save right in stack			
		IF stackCount < 32              					
		THEN                            					
			stackCount 										:= stackCount +1;
		ELSE															// Error stack Limit    
			endMainLoop 									:= TRUE;
			byLTIME											:= FALSE;			
		END_IF                          					
		right 												:= MAX(left, i-1);
	ELSE                                
		IF stackCount = 1 THEN          
			endMainLoop 									:= TRUE;
		ELSE                            					
			left 											:= right+1;       
			stackCount 										:= stackCount -1;	// load from stack
			right											:= TO_DINT(stack[stackCount]);
		END_IF
	END_IF
END_WHILE
END_METHOD

METHOD byREAL : BOOL // returns true if sort ends successfully 
VAR_INPUT
	pData													: 	POINTER TO BYTE := 0;	// ADR(Array) 	
	SizeOfData												: 	UDINT := 0;				// SIZEOF(Array)
	pCompareElement											: 	POINTER TO BYTE := 0;	// ADR(Array[1].REAL)		
	SizeOfStruct											: 	UDINT := 0;				// SIZEOF(Array[1]) 	
END_VAR                                                 
VAR        
	pPivotElement											: 	POINTER TO REAL;		// Pivot value	
	PivotElement											: 	REAL;					// Pivot value as REAL	
	pCmpElement												:	POINTER TO REAL;		// compare value
	                                					                            	
	endMainLoop												:	BOOL;					// End of main loop reached
	endSubLoop												:	BOOL;					// End of sub loop reached                                              
	ElementCount											:	DINT;					// No of array elements
	stackCount,left,right,i,j								:	DINT;					// running variables 	
	stack													:	ARRAY[1..32] OF UDINT;	// stack size 32 => ~1 Mio elements *)	
	                                					
	pElement_1												:	POINTER TO BYTE;		// Copy Pointer 1		
	pElement_2												:	POINTER TO BYTE;		// Copy Pointer 2
END_VAR
// ends with true in case of no error	                                    					 					
IF SizeOfStruct = 0 OR SizeOfData = 0
	OR pData = 0 OR pCompareElement = 0
THEN               					                                   					
	byREAL													:= FALSE;
	RETURN;   
ELSE
	byREAL													:= TRUE;                          					
END_IF                                   					
          
// calculate no. of Elements                                
ElementCount												:= TO_DINT(SizeOfData / SizeOfStruct);   
                              					
// Quicksort                            					
// initial value of array size          					
left 														:= 1;				// first element
right 														:= ElementCount;	// last element 
stackCount 													:= 1;				// running variable 
                                        	
WHILE NOT endMainLoop DO							
	IF left < right THEN                	
		pPivotElement										:= pCompareElement + (SizeOfStruct * TO_UDINT(SHR(right+left,1)));
		PivotElement										:= pPivotElement^;
		i 													:= left -1;
		j 													:= right +1;
		endSubLoop 											:= FALSE;
		REPEAT
			IF SortInverse
			THEN	// sort descending	
				REPEAT	
					i 										:= i+1;	
					pCmpElement								:= pCompareElement + (SizeOfStruct * TO_UDINT(i-1));
				UNTIL (pCmpElement^ <= PivotElement) OR NOT (i < right)	END_REPEAT	
				REPEAT	
					j 										:= j-1;	
					pCmpElement								:= pCompareElement + (SizeOfStruct * TO_UDINT(j-1));
				UNTIL (pCmpElement^ >= PivotElement) OR NOT (j > left)	END_REPEAT		
			ELSE	// sort ascending
				REPEAT	
					i 										:= i+1;
					pCmpElement								:= pCompareElement + (SizeOfStruct * TO_UDINT(i-1));
				UNTIL (pCmpElement^ >= PivotElement)	OR NOT (i < right)	END_REPEAT;				
				REPEAT	
					j 										:= j-1;	
					pCmpElement								:= pCompareElement + (SizeOfStruct * TO_UDINT(j-1));
				UNTIL (pCmpElement^ <= PivotElement) OR NOT (j > left)	END_REPEAT;
			END_IF
			IF i >= j THEN
				endSubLoop									:= TRUE;
			ELSE                    					
				Allocate(SizeOfStruct);
				pElement_1									:= pData + (SizeOfStruct * TO_UDINT(j-1));
				pElement_2									:= pData + (SizeOfStruct * TO_UDINT(i-1));
				
				IF pElement_Tmp = 0 
					OR_ELSE MEMCPY(pElement_Tmp, pElement_1,	SizeOfStruct) = 0
					OR_ELSE MEMCPY(pElement_1,	pElement_2,		SizeOfStruct) = 0
					OR_ELSE MEMCPY(pElement_2,	pElement_Tmp,	SizeOfStruct) = 0
				THEN
					byREAL									:= FALSE;
					RETURN;	
				END_IF

			END_IF
		UNTIL endSubLoop END_REPEAT;		
		stack[stackCount] 									:= TO_UDINT(right); 	// save right in stack			
		IF stackCount < 32              					
		THEN                            					
			stackCount 										:= stackCount +1;
		ELSE															// Error stack Limit    
			endMainLoop 									:= TRUE;
			byREAL											:= FALSE;			
		END_IF                          					
		right 												:= MAX(left, i-1);
	ELSE                                
		IF stackCount = 1 THEN          
			endMainLoop 									:= TRUE;
		ELSE                            					
			left 											:= right+1;       
			stackCount 										:= stackCount -1;	// load from stack
			right											:= TO_DINT(stack[stackCount]);
		END_IF
	END_IF
END_WHILE
END_METHOD

METHOD bySTRING : BOOL // returns true if sort ends successfully 
VAR_INPUT
	pData													: 	POINTER TO BYTE := 0;	// ADR(Array) 	
	SizeOfData												: 	UDINT := 0;				// SIZEOF(Array)
	pCompareElement											: 	POINTER TO BYTE := 0;	// ADR(Array[1].STRING)		
	SizeOfStruct											: 	UDINT := 0;				// SIZEOF(Array[1]) 	
END_VAR                                                                                        
VAR        
	pPivotElement											: 	POINTER TO STRING(MAX_STRING_LENGTH);	// Pivot value
	pCmpElement												:	POINTER TO STRING(MAX_STRING_LENGTH);	// compare value
	PivotElement											:	BYTE; 					// Pivot value	
	CompareElement											:	BYTE; 					// compare value
                               					                            	
